// TwinCAT 3 PLC project Capannone
// ProgramVersion: 3.1.4020.10
// libraries:
//   Tc2_DALI, * (Beckhoff Automation GmbH)
//   Tc2_EnOcean, * (Beckhoff Automation GmbH)
//   Tc2_Standard, * (Beckhoff Automation GmbH)
//   Tc2_SUPS, * (Beckhoff Automation GmbH)
//   Tc2_System, * (Beckhoff Automation GmbH)
//   Tc2_TcpIp, * (Beckhoff Automation GmbH)
//   Tc2_Ulux, * (Beckhoff Automation GmbH Austria)
//   Tc2_Utilities, * (Beckhoff Automation GmbH)
//   Tc3_Module, * (Beckhoff Automation GmbH)
//   TwinCAT PLC Library ekey, * (Beckhoff Automation GmbH Austria)
//   Tc2_EIB,newest,Beckhoff Automation GmbH
//   Tc2_SerialCom,newest,Beckhoff Automation GmbH
// project tree:
//   / Clock_1Sec.TcTTO, PlcTask.TcTTO, Clock_250ms.TcTTO
//   DUTs/ Areotermo.TcDUT, struct_allarme.TcDUT, struct_allarme_1.TcDUT, Struct_Utenti.TcDUT
//   GVLs/ GVL.TcGVL, GVL_ULUX.TcGVL
//   POUs/ ADS_CX8080.TcPOU, Alarm.TcPOU, Clock_5Sec_refresh.TcPOU, Clock_2Sec_refresh_.TcPOU, DALI.TcPOU, Ekey.TcPOU, EnOcean.TcPOU, KNX.TcPOU, LUCI.TcPOU, MAIN.TcPOU, Riscaldamento.TcPOU, Timbrature.TcPOU, TIMER.TcPOU, ULUX.TcPOU
//   POUs/ProjetcFB/ Sensore_Allarme.TcPOU, Dali_arcpower_control.TcPOU, EnO_TK_SR_MDS_BAT.TcPOU, F_COIL.TcPOU, DALI_TK_SR07_rh.TcPOU, DALI_TK_SR07.TcPOU, EnO_TK_SAB05.TcPOU, EnO_TK_SR65_LI.TcPOU, Luci_Mov_Dali.TcPOU, Comando_Luce.TcPOU, Comando_LuceDali.TcPOU, Sensore_Allarme_STRU.TcPOU, Speed_Sabiana.TcPOU, ULUX_STD.TcPOU
// real-time tasks:
//   TASK 10 ms: cycle T#10ms, priority 20, ADS port 350
//   TASK Time250ms: cycle T#250ms, priority 1, ADS port 351
//   TASK Clock_1Sec: cycle T#1000ms, priority 21, ADS port 352
// I/O:
//   DEVICE Device 3 (CX-BK)
//     Box 1 (CX-BK)
//   DEVICE Device 4 (COM Port)
//   DEVICE Device 5 (RT-Ethernet Protocol), AmsNetId 192.168.60.20.6.1
//     I/O Uffici (BK9000)
//     I/O Caldaia (BK9000)
// variable links:
//   Capannone/Capannone Instance <-> Device 3 (CX-BK)/Box 1 (CX-BK)
//     Clock_1Sec Outputs/GVL.Segnale_sirena <-> Term 28 (KL2652)/Channel 2/Output
//     PlcTask Inputs/DALI.DALI_IN1/nData <-> Term 2 (KL6811)/Channel 1/Data In
//     PlcTask Inputs/DALI.DALI_IN1/nStatus <-> Term 2 (KL6811)/Channel 1/State
//     PlcTask Inputs/Ekey.ekey_in/D <-> Term 10 (KL6041)/Channel 1/Data In 0
//     PlcTask Inputs/Ekey.ekey_in/D @bit {8..168 step 8} <-> Term 10 (KL6041)/Channel 1/Data In {1..21}  (21 links)
//     PlcTask Inputs/Ekey.ekey_in/Status <-> Term 10 (KL6041)/Channel 1/State
//     PlcTask Inputs/EnOcean.enocean_in @bit 8 <-> Term 3 (KL6581)/Channel 1/Input CNODE
//     PlcTask Inputs/EnOcean.enocean_in @bit {24..48 step 8} <-> Term 3 (KL6581)/Channel 1/Input DB{0..3}  (4 links)
//     PlcTask Inputs/EnOcean.enocean_in @bit {56..80 step 8} <-> Term 3 (KL6581)/Channel 1/Input ID{0..3}  (4 links)
//     PlcTask Inputs/EnOcean.enocean_in @bit 16 <-> Term 3 (KL6581)/Channel 1/Input ORG
//     PlcTask Inputs/EnOcean.enocean_in @bit 88 <-> Term 3 (KL6581)/Channel 1/Input STATUS
//     PlcTask Inputs/EnOcean.enocean_in <-> Term 3 (KL6581)/Channel 1/Status
//     PlcTask Inputs/GVL.IN_CITOR1 <-> Term 4 (KL1809)/Channel 3/Input
//     PlcTask Inputs/GVL.IN_CITOR2 <-> Term 4 (KL1809)/Channel 2/Input
//     PlcTask Inputs/GVL.SM_C1 <-> Term 27 (KL1809)/Channel 16/Input
//     PlcTask Inputs/GVL.SM_C2 <-> Term 27 (KL1809)/Channel 15/Input
//     PlcTask Inputs/GVL.SM_C3 <-> Term 27 (KL1809)/Channel 14/Input
//     PlcTask Inputs/GVL.SM_F1 <-> Term 4 (KL1809)/Channel 6/Input
//     PlcTask Inputs/GVL.SM_F2 <-> Term 4 (KL1809)/Channel 7/Input
//     PlcTask Inputs/GVL.SM_F3 <-> Term 4 (KL1809)/Channel 8/Input
//     PlcTask Inputs/GVL.SM_F4 <-> Term 4 (KL1809)/Channel 5/Input
//     PlcTask Inputs/GVL.SM_F5 <-> Term 27 (KL1809)/Channel 2/Input
//     PlcTask Inputs/GVL.SM_R2 <-> Term 4 (KL1809)/Channel 15/Input
//     PlcTask Inputs/GVL.SM_R3 <-> Term 4 (KL1809)/Channel 16/Input
//     PlcTask Inputs/GVL.SM_R4 <-> Term 4 (KL1809)/Channel 13/Input
//     PlcTask Inputs/GVL.SM_R5 <-> Term 4 (KL1809)/Channel 14/Input
//     PlcTask Inputs/GVL.SM_S1 <-> Term 27 (KL1809)/Channel 13/Input
//     PlcTask Inputs/GVL.SM_S2 <-> Term 27 (KL1809)/Channel 8/Input
//     PlcTask Inputs/GVL.SM_U1 <-> Term 27 (KL1809)/Channel 5/Input
//     PlcTask Inputs/GVL.SM_U2 <-> Term 27 (KL1809)/Channel 6/Input
//     PlcTask Inputs/GVL.SM_U3 <-> Term 27 (KL1809)/Channel 7/Input
//     PlcTask Inputs/GVL.sens_cancello_Auto <-> Term 4 (KL1809)/Channel 9/Input
//     PlcTask Inputs/MAIN.energy_ch1_dataIN <-> Term 9 (KL3403)/Channel 1/Data In
//     PlcTask Inputs/MAIN.energy_ch2_dataIN <-> Term 9 (KL3403)/Channel 2/Data In
//     PlcTask Inputs/MAIN.energy_ch3_dataIN <-> Term 9 (KL3403)/Channel 3/Data In
//     PlcTask Inputs/MAIN.energy_ch1_state <-> Term 9 (KL3403)/Channel 1/State
//     PlcTask Inputs/MAIN.energy_ch2_state <-> Term 9 (KL3403)/Channel 2/State
//     PlcTask Inputs/MAIN.energy_ch3_state <-> Term 9 (KL3403)/Channel 3/State
//     PlcTask Inputs/MAIN.puls_chiamata <-> Term 4 (KL1809)/Channel 1/Input
//     PlcTask Outputs/DALI.DALI_OUT1/nCtrl <-> Term 2 (KL6811)/Channel 1/Ctrl
//     PlcTask Outputs/DALI.DALI_OUT1/nData <-> Term 2 (KL6811)/Channel 1/Data Out
//     PlcTask Outputs/Ekey.ekey_out/Ctrl <-> Term 10 (KL6041)/Channel 1/Ctrl
//     PlcTask Outputs/Ekey.ekey_out/D <-> Term 10 (KL6041)/Channel 1/Data Out 0
//     PlcTask Outputs/Ekey.ekey_out/D @bit {8..168 step 8} <-> Term 10 (KL6041)/Channel 1/Data Out {1..21}  (21 links)
//     PlcTask Outputs/EnOcean.enocean_out <-> Term 3 (KL6581)/Channel 1/Control
//     PlcTask Outputs/EnOcean.enocean_out @bit 8 <-> Term 3 (KL6581)/Channel 1/Output CNODE
//     PlcTask Outputs/EnOcean.enocean_out @bit {24..48 step 8} <-> Term 3 (KL6581)/Channel 1/Output DB{0..3}  (4 links)
//     PlcTask Outputs/EnOcean.enocean_out @bit {56..80 step 8} <-> Term 3 (KL6581)/Channel 1/Output ID{0..3}  (4 links)
//     PlcTask Outputs/EnOcean.enocean_out @bit 16 <-> Term 3 (KL6581)/Channel 1/Output ORG
//     PlcTask Outputs/EnOcean.enocean_out @bit 88 <-> Term 3 (KL6581)/Channel 1/Output STATUS
//     PlcTask Outputs/GVL.OUT_Pcanc_ped <-> Term 5 (KL2809)/Channel 2/Output
//     PlcTask Outputs/GVL.Sabiana{1..6}H <-> Term 12 (KL2809)/Channel {1..11 step 2}/Output  (6 links)
//     PlcTask Outputs/GVL.Sabiana{1..6}L <-> Term 12 (KL2809)/Channel {2..12 step 2}/Output  (6 links)
//     PlcTask Outputs/GVL.Segnale_radio <-> Term 28 (KL2652)/Channel 1/Output
//     PlcTask Outputs/LUCI.luci_esterne <-> Term 5 (KL2809)/Channel 5/Output
//     PlcTask Outputs/MAIN.apert_canc <-> Term 5 (KL2809)/Channel 1/Output
//     PlcTask Outputs/MAIN.compr_pistone <-> Term 5 (KL2809)/Channel 7/Output
//     PlcTask Outputs/MAIN.compr_vite <-> Term 5 (KL2809)/Channel 8/Output
//     PlcTask Outputs/MAIN.energy_ch1_control <-> Term 9 (KL3403)/Channel 1/Ctrl
//     PlcTask Outputs/MAIN.energy_ch2_control <-> Term 9 (KL3403)/Channel 2/Ctrl
//     PlcTask Outputs/MAIN.energy_ch3_control <-> Term 9 (KL3403)/Channel 3/Ctrl
//     PlcTask Outputs/MAIN.sirena_canc <-> Term 7 (KL2602)/Channel 1/Output
//   Capannone/Capannone Instance <-> Device 5 (RT-Ethernet Protocol)/I/O Caldaia (BK9000)
//     PlcTask Inputs/Riscaldamento.run_pompaprod <-> Term 39 (KL1002)/Channel 1/Input
//     PlcTask Inputs/Riscaldamento.temp_ciller <-> Term 40 (KL3204)/Channel 1/Data In
//     PlcTask Outputs/Riscaldamento.pompa_prod1 <-> Term 41 (KM2642)/Channel 1/Output
//     PlcTask Outputs/Riscaldamento.pompa_prod2 <-> Term 42 (KM2642)/Channel 2/Output
//     PlcTask Outputs/Riscaldamento.richiesta_caldaia <-> Term 42 (KM2642)/Channel 1/Output
//   Capannone/Capannone Instance <-> Device 5 (RT-Ethernet Protocol)/I/O Uffici (BK9000)
//     Clock_1Sec Outputs/GVL.Luce5 <-> Term 20 (KL2809)/Channel 5/Output
//     Clock_1Sec Outputs/GVL.Luce6 <-> Term 20 (KL2809)/Channel 6/Output
//     PlcTask Inputs/DALI.DALI_IN2/nData <-> Term 14 (KL6811)/Channel 1/Data In
//     PlcTask Inputs/DALI.DALI_IN2/nStatus <-> Term 14 (KL6811)/Channel 1/State
//     PlcTask Inputs/GVL.Th20_pompacaloreOK <-> Term 15 (KL1809)/Channel 2/Input
//     PlcTask Inputs/GVL.pulA1 <-> Term 15 (KL1809)/Channel 5/Input
//     PlcTask Inputs/GVL.pulA2 <-> Term 15 (KL1809)/Channel 3/Input
//     PlcTask Inputs/GVL.pulA3 <-> Term 15 (KL1809)/Channel 6/Input
//     PlcTask Inputs/GVL.pulA4 <-> Term 15 (KL1809)/Channel 4/Input
//     PlcTask Inputs/GVL.pulB1 <-> Term 15 (KL1809)/Channel 8/Input
//     PlcTask Inputs/GVL.pulB2 <-> Term 15 (KL1809)/Channel 7/Input
//     PlcTask Inputs/GVL.pulC1 <-> Term 15 (KL1809)/Channel 9/Input
//     PlcTask Inputs/GVL.pulD1 <-> Term 15 (KL1809)/Channel 10/Input
//     PlcTask Inputs/KNX.KNX_IN @bit {16..184 step 8} <-> Term 21 (KL6301)/Channel 1/Input Data {1..22}  (22 links)
//     PlcTask Inputs/KNX.KNX_IN <-> Term 21 (KL6301)/Channel 1/Parameter Status
//     PlcTask Outputs/DALI.DALI_OUT2/nCtrl <-> Term 14 (KL6811)/Channel 1/Ctrl
//     PlcTask Outputs/DALI.DALI_OUT2/nData <-> Term 14 (KL6811)/Channel 1/Data Out
//     PlcTask Outputs/GVL.Aer_Bagni <-> Term 20 (KL2809)/Channel 8/Output
//     PlcTask Outputs/GVL.Aer_Uffici <-> Term 20 (KL2809)/Channel 7/Output
//     PlcTask Outputs/GVL.Luce{1..4} <-> Term 20 (KL2809)/Channel {1..4}/Output  (4 links)
//     PlcTask Outputs/GVL.OUT_CILLER_ON <-> Term 19 (KL2809)/Channel 6/Output
//     PlcTask Outputs/GVL.OUT_Pingresso <-> Term 19 (KL2809)/Channel 3/Output
//     PlcTask Outputs/GVL.OUT_Pmensa <-> Term 19 (KL2809)/Channel 4/Output
//     PlcTask Outputs/GVL.out_ciller_estate <-> Term 19 (KL2809)/Channel 5/Output
//     PlcTask Outputs/KNX.KNX_OUT @bit {16..184 step 8} <-> Term 21 (KL6301)/Channel 1/Output Data {1..22}  (22 links)
//     PlcTask Outputs/KNX.KNX_OUT <-> Term 21 (KL6301)/Channel 1/Parameter Control
//     PlcTask Outputs/Riscaldamento.areotermi[10]/VHL1 <-> Term 19 (KL2809)/Channel 1/Output
//     PlcTask Outputs/Riscaldamento.areotermi[10]/VHL2 <-> Term 19 (KL2809)/Channel 2/Output
//     PlcTask Outputs/Riscaldamento.areotermi[1]/VHL1 <-> Term 16 (KL2809)/Channel 4/Output
//     PlcTask Outputs/Riscaldamento.areotermi[1]/VHL2 <-> Term 16 (KL2809)/Channel 5/Output
//     PlcTask Outputs/Riscaldamento.areotermi[2]/VHL1 <-> Term 16 (KL2809)/Channel 9/Output
//     PlcTask Outputs/Riscaldamento.areotermi[2]/VHL2 <-> Term 16 (KL2809)/Channel 10/Output
//     PlcTask Outputs/Riscaldamento.areotermi[3]/VHL1 <-> Term 16 (KL2809)/Channel 14/Output
//     PlcTask Outputs/Riscaldamento.areotermi[3]/VHL2 <-> Term 16 (KL2809)/Channel 15/Output
//     PlcTask Outputs/Riscaldamento.areotermi[4]/VHL1 <-> Term 17 (KL2809)/Channel 3/Output
//     PlcTask Outputs/Riscaldamento.areotermi[4]/VHL2 <-> Term 17 (KL2809)/Channel 4/Output
//     PlcTask Outputs/Riscaldamento.areotermi[5]/VHL1 <-> Term 17 (KL2809)/Channel 8/Output
//     PlcTask Outputs/Riscaldamento.areotermi[5]/VHL2 <-> Term 17 (KL2809)/Channel 9/Output
//     PlcTask Outputs/Riscaldamento.areotermi[6]/VHL1 <-> Term 17 (KL2809)/Channel 13/Output
//     PlcTask Outputs/Riscaldamento.areotermi[6]/VHL2 <-> Term 17 (KL2809)/Channel 14/Output
//     PlcTask Outputs/Riscaldamento.areotermi[7]/VHL1 <-> Term 18 (KL2809)/Channel 2/Output
//     PlcTask Outputs/Riscaldamento.areotermi[7]/VHL2 <-> Term 18 (KL2809)/Channel 3/Output
//     PlcTask Outputs/Riscaldamento.areotermi[8]/VHL1 <-> Term 18 (KL2809)/Channel 7/Output
//     PlcTask Outputs/Riscaldamento.areotermi[8]/VHL2 <-> Term 18 (KL2809)/Channel 8/Output
//     PlcTask Outputs/Riscaldamento.areotermi[9]/VHL1 <-> Term 18 (KL2809)/Channel 12/Output
//     PlcTask Outputs/Riscaldamento.areotermi[9]/VHL2 <-> Term 18 (KL2809)/Channel 13/Output
//     PlcTask Outputs/Riscaldamento.areotermi[10]/speed1 <-> Term 18 (KL2809)/Channel 14/Output
//     PlcTask Outputs/Riscaldamento.areotermi[10]/speed2 <-> Term 18 (KL2809)/Channel 15/Output
//     PlcTask Outputs/Riscaldamento.areotermi[10]/speed3 <-> Term 18 (KL2809)/Channel 16/Output
//     PlcTask Outputs/Riscaldamento.areotermi[1]/speed1 <-> Term 16 (KL2809)/Channel 1/Output
//     PlcTask Outputs/Riscaldamento.areotermi[1]/speed2 <-> Term 16 (KL2809)/Channel 2/Output
//     PlcTask Outputs/Riscaldamento.areotermi[1]/speed3 <-> Term 16 (KL2809)/Channel 3/Output
//     PlcTask Outputs/Riscaldamento.areotermi[2]/speed1 <-> Term 16 (KL2809)/Channel 6/Output
//     PlcTask Outputs/Riscaldamento.areotermi[2]/speed2 <-> Term 16 (KL2809)/Channel 7/Output
//     PlcTask Outputs/Riscaldamento.areotermi[2]/speed3 <-> Term 16 (KL2809)/Channel 8/Output
//     PlcTask Outputs/Riscaldamento.areotermi[3]/speed1 <-> Term 16 (KL2809)/Channel 11/Output
//     PlcTask Outputs/Riscaldamento.areotermi[3]/speed2 <-> Term 16 (KL2809)/Channel 12/Output
//     PlcTask Outputs/Riscaldamento.areotermi[3]/speed3 <-> Term 16 (KL2809)/Channel 13/Output
//     PlcTask Outputs/Riscaldamento.areotermi[4]/speed1 <-> Term 16 (KL2809)/Channel 16/Output
//     PlcTask Outputs/Riscaldamento.areotermi[4]/speed2 <-> Term 17 (KL2809)/Channel 1/Output
//     PlcTask Outputs/Riscaldamento.areotermi[4]/speed3 <-> Term 17 (KL2809)/Channel 2/Output
//     PlcTask Outputs/Riscaldamento.areotermi[5]/speed1 <-> Term 17 (KL2809)/Channel 5/Output
//     PlcTask Outputs/Riscaldamento.areotermi[5]/speed2 <-> Term 17 (KL2809)/Channel 6/Output
//     PlcTask Outputs/Riscaldamento.areotermi[5]/speed3 <-> Term 17 (KL2809)/Channel 7/Output
//     PlcTask Outputs/Riscaldamento.areotermi[6]/speed1 <-> Term 17 (KL2809)/Channel 10/Output
//     PlcTask Outputs/Riscaldamento.areotermi[6]/speed2 <-> Term 17 (KL2809)/Channel 11/Output
//     PlcTask Outputs/Riscaldamento.areotermi[6]/speed3 <-> Term 17 (KL2809)/Channel 12/Output
//     PlcTask Outputs/Riscaldamento.areotermi[7]/speed1 <-> Term 17 (KL2809)/Channel 15/Output
//     PlcTask Outputs/Riscaldamento.areotermi[7]/speed2 <-> Term 17 (KL2809)/Channel 16/Output
//     PlcTask Outputs/Riscaldamento.areotermi[7]/speed3 <-> Term 18 (KL2809)/Channel 1/Output
//     PlcTask Outputs/Riscaldamento.areotermi[8]/speed1 <-> Term 18 (KL2809)/Channel 4/Output
//     PlcTask Outputs/Riscaldamento.areotermi[8]/speed2 <-> Term 18 (KL2809)/Channel 5/Output
//     PlcTask Outputs/Riscaldamento.areotermi[8]/speed3 <-> Term 18 (KL2809)/Channel 6/Output
//     PlcTask Outputs/Riscaldamento.areotermi[9]/speed1 <-> Term 18 (KL2809)/Channel 9/Output
//     PlcTask Outputs/Riscaldamento.areotermi[9]/speed2 <-> Term 18 (KL2809)/Channel 10/Output
//     PlcTask Outputs/Riscaldamento.areotermi[9]/speed3 <-> Term 18 (KL2809)/Channel 11/Output

CONFIGURATION Capannone
    RESOURCE PLC ON TwinCAT3
        TASK Clock_1Sec(INTERVAL := T#1000ms, PRIORITY := 21);
        TASK PlcTask(INTERVAL := T#10ms, PRIORITY := 20);
        TASK Clock_250ms(INTERVAL := T#250ms, PRIORITY := 1);
        PROGRAM Clock_5Sec_refresh WITH Clock_1Sec : Clock_5Sec_refresh;
        PROGRAM Clock_2Sec_refresh_ WITH Clock_1Sec : Clock_2Sec_refresh_;
        PROGRAM MAIN WITH PlcTask : MAIN;
        PROGRAM Timbrature WITH PlcTask : Timbrature;
        PROGRAM TIMER WITH Clock_250ms : TIMER;
    END_RESOURCE
END_CONFIGURATION

// ---- DUTs/Areotermo.TcDUT
TYPE Areotermo :
STRUCT
	speed1:BOOL;
	speed2:BOOL;
	speed3:BOOL;
	VHL1:BOOL;
	VHL2:BOOL;
END_STRUCT
END_TYPE

// ---- DUTs/struct_allarme.TcDUT
TYPE struct_allarme :
STRUCT
	mode_a0 : BOOL:=TRUE;
	mode_a1 : BOOL;
	mode_a2 : BOOL;
	mode_a3 : BOOL;
	mode_a4 : BOOL;
	delay_allarme : TIME:= T#30S;
	allarme_dis : BOOL;
	sens_mov : BOOL;
	porta_fin : BOOL;
	sensore : BOOL;
	sens_ritardato : BOOL;
	sens_attivo : BOOL;
END_STRUCT
END_TYPE

// ---- DUTs/struct_allarme_1.TcDUT
TYPE struct_allarme_1 :
STRUCT
	sens_zonaA: BOOL;
	sens_zonaB: BOOL;
	sens_zonaC: BOOL;
	sens_zonaD: BOOL;
	ritardo_ON: TIME; //Ritardo accensione sensore in secondi
	ritardo_OFF: TIME; //Ritardo spegnimento sensore in secondi
	HMI_Ritardo_ON: REAL; //HMI ritardo accensione sensore
	HMI_Ritardo_OFF: REAL; //HMI ritardo spegnimento sensore
	sens_ON_OFF: BOOL; //Accensione/spegnimento sensore TRUE=acceso FALSE= spento
	allarme_sensore: BOOL; //Segnale uscita allarme sensore
	tamper_sensore: BOOL; //Segnale uscita tamper sensore
	stato_sensore: BYTE; //0=OFF 1=allarme generato 2=tamper 3=in allarme attivo ma libero 4=in allarme attivo 5=acceso libero 6=acceso occupato
	testo_sensore: STRING; //Nome e funzione sensore
	sensore_preallarme: BOOL; //Segnale sonoro con allarme attivo
END_STRUCT
END_TYPE

// ---- DUTs/Struct_Utenti.TcDUT
TYPE Struct_Utenti :
STRUCT
	user_type: BYTE;
	num_badge: STRING;
	nome_utente: STRING;
END_STRUCT
END_TYPE

// ---- GVLs/GVL.TcGVL
VAR_GLOBAL
	//cancella
	AAA_Prova1: BOOL;
	//EnOcean
	enocean_buffer: STR_KL6581;
	//DALI
	DALI_BUFFER1: ST_DALIV2CommandBuffer; //Comando luci capannone
	DALI_BUFFER2: ST_DALIV2CommandBuffer; //Comando luci uffici
	//Ekey
	ekey_scanner_cancello: FB_EKEY_FingerScanner; //Numero di serie ekey cancello:31160073
	ekey_scanner_produzione: FB_EKEY_FingerScanner; //Numero di serie ekey produzione:24180820 vecchio:37160686
	ekey_scanner_ingresso: FB_EKEY_FingerScanner;//Numero di serie ekey ingresso:37160693 vecchio:37160693
	HMI_finger: BOOL;
	HMI_finger_RFID: BOOL;
	HMI_userRFID: BYTE;
	apri_file: FB_FileOpen;
	inserisci_testo: fb_fileputs;
	chiudi_file: fb_fileclose;
	indice_utente: INT:=1;
	Nmu: BYTE:=30; //Numero massimo utenti
	hmi_utentesu: BOOL; //Pulsante indice utente i più
	hmi_utentegiu: BOOL; //Pulsante indice utente i meno
	HMI_save_utente: BOOL; //Salva parametri utenti su HMI
	HMI_annulla: BOOL; // Annulla cambio dati utente
	HMI_user_type: BYTE;
	HMI_num_badge: STRING;
	HMI_nome_utente: STRING;
	//ULUX
	ulux_buffer: ST_ULUX_COMMANDBUFFER;
	//KNX
	RAIN: BOOL;
	Temp_OUTSIDE: REAL;
	wind_speed: REAL;
	LUX_OUTSIDEF: REAL;
	LUX_OUTSIDER: REAL;
	LUX_OUTSIDEL: REAL;
	knx_p1: BOOL;
	knx_p2: BOOL;
	knx_p3: BOOL;
	knx_p4: BOOL;
	Temp_INSIDE: REAL;
	stato_temp: BOOL; //Stato sensore temperatura 0=OK 1=Difettoso
	
	//ALLARME
	alarm_Service: BOOL;
	allarme_on: BOOL;
	sensori_mov: ARRAY [1..30] OF sensore_allarme;
	mode_A: BYTE; //Modalità inserimento allarme valori da 0 a 4
	test_Sirena: BOOL;
	test_radio: BOOL;
	allarme_memreset: BOOL;
	stringa_allarme: STRING;
	stringa_2_allarme: STRING; //Stringa di visualizzazione in file di testo allarmi
	sensori_STRU: ARRAY [0..30] OF sensore_allarme_STRU;
	ingresso_sens AT %I*: ARRAY [0..30] OF BOOL; //Array segnale fisico sensore
	reset_tamper: BOOL;
	reset_allarme: BOOL;
	manutenzione_sensore: BOOL;
	
	//CILLER
	out_ciller_estate AT %Q*: BOOL;
	OUT_CILLER_ON AT %Q*: BOOL;
	//PORTE
	OUT_Pingresso AT %Q*: BOOL;
	OUT_Pmensa AT %Q*: BOOL;
	OUT_Pcanc_ped AT %Q*: BOOL;
	IN_CITOR1 AT %I*: BOOL;
	IN_CITOR2 AT %I*: BOOL;
	//ALTRO
	tempo: BOOL;
	count: INT;
	ora_plc: nt_gettime;
	tempo_ulux: timestruct;
	aggiorna: BYTE; //Variabile timer
	orario: STRING;
	orario_2: STRING;
	giorni_sett: BOOL;
	Read_Puls1: FB_Rec_RPS_Switch;
	HMI_ctrl_allarme: BOOL;
	sens_cancello_Auto AT %I*: BOOL;
	hmi_cancello: BOOL;
	HMI_compressore_2: BOOL;
	HMI_currentL1: WORD;
	HMI_currentL2: WORD;
	HMI_currentL3: WORD;
	HMI_voltageL1: WORD;
	HMI_voltageL2: WORD;
	HMI_voltageL3: WORD;
	HMI_powerL1: WORD;
	HMI_powerL2: WORD;
	HMI_powerL3: WORD;
	HMI_energyL1: WORD;
	HMI_energyL2: WORD;
	HMI_energyL3: WORD;
	HMI_frequencyL1: WORD;
	HMI_frequencyL2: WORD;
	HMI_frequencyL3: WORD;
	HMI_Allarme: BOOL;
	HMI_luci_on: ARRAY [0..6] OF BOOL; //Luci uffici ON
	HMI_luci_off: ARRAY [0..6] OF BOOL; //Luci uffici OFF
	HMI_cond: ARRAY [0..6] OF INT;
	HMI_luce1: BOOL; //Comando luce bagno 1 da HMI
	HMI_luce2: BOOL; //Comando luce bagno 2 da HMI
	HMI_luce_3: BOOL; //Comando luci esterne da HMI
	HMI_luce4: BOOL; //Comando luce ripostiglio da HMI
	HMI_luce_server: BOOL; //Comando luce server da HMI
	HMI_luce_lstamp: BOOL; //Comando luce locale stampante
	HMI_luce_offRD: BOOL; //Comando luce officina R&D
	
	light_soft: BOOL;
	Light_on: BOOL;
	Light_off: BOOL;
	dali_power_off: BOOL;
	Sabiana1L AT %Q*: BOOL; //Sabiana 1 Low Speed
	Sabiana1H AT %Q*: BOOL; //Sabiana 1 High Speed
	Sabiana2L AT %Q*: BOOL; //Sabiana 2 Low Speed
	Sabiana2H AT %Q*: BOOL; //Sabiana 2 High Speed
	Sabiana3L AT %Q*: BOOL; //Sabiana 3 Low Speed
	Sabiana3H AT %Q*: BOOL; //Sabiana 3 High Speed
	Sabiana4L AT %Q*: BOOL; //Sabiana 4 Low Speed
	Sabiana4H AT %Q*: BOOL; //Sabiana 4 High Speed
	Sabiana5L AT %Q*: BOOL; //Sabiana 5 Low Speed
	Sabiana5H AT %Q*: BOOL; //Sabiana 5 High Speed
	Sabiana6L AT %Q*: BOOL; //Sabiana 6 Low Speed
	Sabiana6H AT %Q*: BOOL; //Sabiana 6 High Speed
	
	HMI_SabianaManCTRL : ARRAY [1..6] OF BYTE; //Controllo Manuale Sabiana
	HMI_PompaProd : BOOL; //Comando Manuale da pannello pompa riscaldamento produzione
	TempZ0:UINT; //Temperatura zona 0 - Capannone
	TempZ1:UINT; //Temperatura zona 1 - Ingresso
	TempZ2:UINT; //Temperatura zona 2 - Amministrazione
	TempZ3:UINT; //Temperatura zona 3 - Direzione
	TempZ4:UINT; //Temperatura zona 4 - Sala Riunioni
	TempZ5:UINT; //Temperatura zona 5 - Uffico Tecnico
	TempZ6:UINT; //Temperatura zona 6 - Ufficio Produzione
	TempZ7:UINT; //Temperatura zona 7 - Locale Svago
	ConONz1:INT; //Condizionatore ON/OFF zona 1
	ConONz2:INT; //Condizionatore ON/OFF zona 2
	ConONz3:INT; //Condizionatore ON/OFF zona 3
	ConONz4:INT; //Condizionatore ON/OFF zona 4
	ConONz5:INT; //Condizionatore ON/OFF zona 5
	ConONz6:INT; //Condizionatore ON/OFF zona 6
	ConONz7:INT; //Condizionatore ON/OFF zona 7
	HMI_Umidita:BYTE; //Umidità Capannone
	Th20_CaldaiaOK (*AT %I**):BOOL:=TRUE; //Temperatura H20 Caldaia OK x aria
	Th20_pompacaloreOK AT %I*:BOOL; //Temperatura H20 Pompa Calore OK x aria
	SensoreSez1 : BOOL; (*Sensore Apertura Sezionale 1*)
	SensoreSez2 : BOOL; (*Sensore Apertura Sezionale 2*)
	Luce1 AT %Q*:BOOL; (*Relè Luci BAGNO UFFICI 1*)
	Luce2 AT %Q*:BOOL; (*Relè Luci BAGNO UFFICI 2*)
	Luce3 AT %Q*:BOOL; (*Relè Luci esterno ENTRATA*)
	Luce4 AT %Q*:BOOL; (*Relè Luci RIPOSTIGLIO*)
	Luce5 AT %Q*:BOOL; (*Relè Luci 1*)
	Luce6 AT %Q*:BOOL; (*Relè Luci 1*)
	Aer_Uffici AT %Q*:BOOL; (*Relè Luci 1*)
	Aer_Bagni AT %Q* :BOOL; (*Areazione Bagno*)
	time_now: UINT;
	GuestIN_OK: BOOL;
	UserIN_OK: BOOL;
	HMI_blink: BOOL; //Bit per blink su HMI
	luci_ufficio_off: BOOL;
	//Pulsantiera A
	pulA1 AT %I* :BOOL;
	pulA2 AT %I* :BOOL;
	pulA3 AT %I* :BOOL;
	pulA4 AT %I* :BOOL;
	//Pulsantiera B
	pulB1 AT %I* :BOOL;
	pulB2 AT %I* :BOOL;
	//Pulsantiera C
	pulC1 AT %I* :BOOL;
	//Pulsantiera D
	pulD1 AT %I* :BOOL;
	prod_summer_fan: INT;
	meetingroom_active: BOOL;
	//Sensori di movimento
	SM_F1 AT %I*: BOOL;
	SM_F2 AT %I*: BOOL;
	SM_F3 AT %I*: BOOL;
	SM_F4 AT %I*: BOOL;
	SM_F5 AT %I*: BOOL;
	SM_S1 AT %I*: BOOL;
	SM_S2 AT %I*: BOOL;
	(*SM_R1 AT %I*: BOOL;
	SM_R2 AT %I*: BOOL;
	SM_R3 AT %I*: BOOL;
	SM_R4 AT %I*: BOOL;
	SM_R5 AT %I*: BOOL;
	SM_D1 AT %I*: BOOL;*)
	SM_C1 AT %I*: BOOL;
	//SM_C2 AT %I*: BOOL;
	//SM_C3 AT %I*: BOOL;
	SM_U1 AT %I*: BOOL; //Sensore Ufficio Tecnico
	SM_U2 AT %I*: BOOL; //Sensore Locale Svago
	//SM_U3 AT %I*: BOOL; //Sensore Ingresso
	Tamper_interno AT %I*: BOOL;
	Tamper_fronte AT %I*: BOOL;
	Tamper_retro AT %I*: BOOL;
	Tamper_sinistro AT %I*: BOOL;
	Segnale_radio AT %Q*: BOOL;
	Segnale_sirena AT %Q*: BOOL;
	
	OFFICE_vhac_MODE:BYTE; //0= ESTATE - 1 INVERNO PDC - 2 INVERNO MISTO
	gruppo8_arc_level: BYTE;
	gruppo9_arc_level: BYTE;
	//Telecamere
	camera_index: INT;
	HMI_blink_2: BOOL;
	HMI_Cancelletto: BOOL;
	HMI_porta: BOOL;
	camera_counter: INT;
	str_camera1: STRING(255);
	camera1: STRING(255);
	camera2: STRING(255);
	camera3: STRING(255);
	camera4: STRING(255);
	//Comando luci bagno produzione e spogliatoi
	count_bagno_prod: INT;
	timer_bagno_prod: TP;
	pulse_bagno_prod: TP;
	luce_bagni: FB_Send_RPS_SwitchAuto;
	luce_spogliatoio: FB_Send_RPS_SwitchAuto;
	MOVIMENTO_BAGNO_PROD: EnO_TK_SR_MDS_BAT;
	RITARDO_LUCE_BAGNO_PROD: TOF;
	
	variable_update: BOOL := FALSE;
	aggiorna_sec: BOOL;
END_VAR
VAR_GLOBAL RETAIN PERSISTENT
	ON:BOOL := TRUE;
	var_ora_trasp: BOOL;
	var_ora_dip: BOOL;
	user_type: ARRAY [1..30] OF BYTE;
	utenti: ARRAY [1..30] OF struct_utenti;
	allarme: BOOL;
	allarme_Attivo: BYTE; //0=OFF 1=Gruppo A 2=Gruppo B 3=Gruppo C 4=Gruppo D
	HMI_sirena: BOOL; //Per ON-OFF segnale sirena da HMI
	HMI_radio: BOOL; //Per ON-OFF segnale radio da HMI
	delay_allarme_on: TIME:=T#150S;
	delay_sirena_off: TIME:=T#2M;
	time_IN1:UINT:=0630;
	time_OUT1:UINT:=1300;
	time_IN2:UINT:=1300;
	time_out2:UINT:=1800;
	time_work_IN1:UINT:=0800;
	time_work_OUT1:UINT:=1230;
	time_work_IN2:UINT:=1330;
	time_work_OUT2:UINT:=1700;
	saturday_work:BOOL;
	holidays:BOOL;
	auto_allarm: BOOL:=TRUE;
	HeatingdMode : BYTE := 2; (*Modo funzionamento riscaldamento 0= OFF - 1=MAN - 2=AUTO - 3=Estate*)
	OFFICE_VHAC_EI:BOOL; (*0=INVERNO 1=ESTATE*)
	estate: BOOL;
	inverno: BOOL;
	HMI_TEMPprod : UINT:=170; (*Temperatura di riferimento PRODUZIONE*)
	HMI_TEMPuff : ARRAY [1..7] OF UINT; //Array temperatura di riferimento UFFICI tec. e prod. è la stessa
	HMI_var_tempuff : ARRAY [1..7] OF UINT; //Array variazione temperatura ambiente UFFICI
	HMI_TEMPuff_max: UINT:=280; //Temperatura di riferimento massima UFFICI
	HMI_TEMPuff_min: UINT:=240; //Temperatura di riferimento minima UFFICI
	HMI_luci_capannone: BYTE:=250; (*Luminosità luci capannone*)
	luci_capannone_aut: BOOL:=TRUE;
	sens_allarme: ARRAY [1..30] OF struct_allarme;
	sens_allarme_stru: ARRAY [0..30] OF struct_allarme_1; //Array struttura sensori
	tamper AT %I*: ARRAY [0..30] OF BOOL; //Array segnale tamper sensore
	alarm_history: ARRAY [1..50] OF STRING;
	warning_history: ARRAY [1..50] OF STRING;
	
	TempOffSabiana1: INT:=450; (*Temperatura Ciller OFF x Sabiana*)
	TempOffSabiana2: INT:=450; (*Temperatura Ciller OFF x Sabiana*)
	TempOffSabiana3: INT:=650; (*Temperatura Ciller OFF x Sabiana*)
	TempOffSabiana4: INT:=550; (*Temperatura Ciller OFF x Sabiana*)
	TempOffSabiana5: INT:=450; (*Temperatura Ciller OFF x Sabiana*)
	TempOffSabiana6: INT:=600; (*Temperatura Ciller OFF x Sabiana*)
END_VAR

// ---- GVLs/GVL_ULUX.TcGVL
(* Automatic generated on 16/02/2017 16.07.46 from u::Lux Config V1.34.635, Build 2474 *)
(* u::Lux Projectfile: C:\Users\ACO\Documents\OWNCLOUD\Software PLC\00 - DOMOTICA\4 - ULUX\Programma_Uffici.uLux *)

(* VarNameEndings: *)
(* _IP: IP-Address of a Control or a Switch *)
(* _ID: ID of an Actor or a Switch *)
(* _EDITVALUE: EditValue of an Actor *)
(* _OUTPUT: Output of an Actor *)
(* _INPUT: Input of an Actor *)

VAR_GLOBAL CONSTANT
	(* Common Constants *)
	PROJEKT_ULUX_CONTROL_IP:STRING:='192.168.60.120';
	PROJEKT_ULUX_CONTROL_AMSNETID:STRING:= '5.29.125.252.1.1';

	(* Constants for u::Lux Switch Design_Ingresso *)
	ULUX_SWITCH_DESIGN_INGRESSO_ULUX_SWITCH_INGRESSO_ID:WORD:=1;

	(* Constants for u::Lux Switch Design_Ingresso\Attori_Ingresso *)
	ATTORI_INGRESSO_ONOFF_LUCE_ID:WORD:=1;
	ATTORI_INGRESSO_DIMMER_ID:WORD:=2;
	ATTORI_INGRESSO_HEIZUNG_TEMPERATUR_ID:WORD:=3;
	ATTORI_INGRESSO_ACTOR_4_ID:WORD:=4;
	ATTORI_INGRESSO_COND_ONOFF_ID:WORD:=5;
	ATTORI_INGRESSO_ACTOR_6_ID:WORD:=6;
	ATTORI_INGRESSO_ACTOR_7_ID:WORD:=7;
	ATTORI_INGRESSO_ACTOR_8_ID:WORD:=8;
	ATTORI_INGRESSO_ACTOR_9_ID:WORD:=9;
	ATTORI_INGRESSO_ACTOR_10_ID:WORD:=10;

	(* Constants for u::Lux Switch Design_Amministrazione *)
	ULUX_SWITCH_DESIGN_AMMINISTRAZIONE_ULUX_SWITCH_AMMINISTRAZIONE_ID:WORD:=2;

	(* Constants for u::Lux Switch Design_Amministrazione\Attori_Amministrazione *)
	ATTORI_AMMINISTRAZIONE_ONOFF_LUCE_ID:WORD:=11;
	ATTORI_AMMINISTRAZIONE_DIMMER_ID:WORD:=12;
	ATTORI_AMMINISTRAZIONE_HEIZUNG_TEMPERATUR_ID:WORD:=13;
	ATTORI_AMMINISTRAZIONE_ACTOR_4_ID:WORD:=14;
	ATTORI_AMMINISTRAZIONE_COND_ONOFF_ID:WORD:=15;
	ATTORI_AMMINISTRAZIONE_ACTOR_6_ID:WORD:=16;
	ATTORI_AMMINISTRAZIONE_ACTOR_7_ID:WORD:=17;
	ATTORI_AMMINISTRAZIONE_ACTOR_8_ID:WORD:=18;
	ATTORI_AMMINISTRAZIONE_ACTOR_9_ID:WORD:=19;
	ATTORI_AMMINISTRAZIONE_ACTOR_10_ID:WORD:=20;

	(* Constants for u::Lux Switch Design_Direzione *)
	ULUX_SWITCH_DESIGN_DIREZIONE_ULUX_SWITCH_DIREZIONE_ID:WORD:=3;

	(* Constants for u::Lux Switch Design_Direzione\Attori_Direzione *)
	ATTORI_DIREZIONE_ONOFF_LUCE_ID:WORD:=21;
	ATTORI_DIREZIONE_DIMMER_ID:WORD:=22;
	ATTORI_DIREZIONE_HEIZUNG_TEMPERATUR_ID:WORD:=23;
	ATTORI_DIREZIONE_ACTOR_4_ID:WORD:=24;
	ATTORI_DIREZIONE_COND_ONOFF_ID:WORD:=25;
	ATTORI_DIREZIONE_ACTOR_6_ID:WORD:=26;
	ATTORI_DIREZIONE_ACTOR_7_ID:WORD:=27;
	ATTORI_DIREZIONE_ACTOR_8_ID:WORD:=28;
	ATTORI_DIREZIONE_ACTOR_9_ID:WORD:=29;
	ATTORI_DIREZIONE_ACTOR_10_ID:WORD:=30;

	(* Constants for u::Lux Switch Design_Sala_Riunioni *)
	ULUX_SWITCH_DESIGN_SALA_RIUNIONI_ULUX_SWITCH_SALA_RIUNIONI_ID:WORD:=4;

	(* Constants for u::Lux Switch Design_Sala_Riunioni\Attori_Sala_Riunioni *)
	ATTORI_SALA_RIUNIONI_ONOFF_LUCE_ID:WORD:=31;
	ATTORI_SALA_RIUNIONI_DIMMER_ID:WORD:=32;
	ATTORI_SALA_RIUNIONI_HEIZUNG_TEMPERATUR_ID:WORD:=33;
	ATTORI_SALA_RIUNIONI_ACTOR_4_ID:WORD:=34;
	ATTORI_SALA_RIUNIONI_COND_ONOFF_ID:WORD:=35;
	ATTORI_SALA_RIUNIONI_ACTOR_6_ID:WORD:=36;
	ATTORI_SALA_RIUNIONI_ACTOR_7_ID:WORD:=37;
	ATTORI_SALA_RIUNIONI_ACTOR_8_ID:WORD:=38;
	ATTORI_SALA_RIUNIONI_ACTOR_9_ID:WORD:=39;
	ATTORI_SALA_RIUNIONI_ACTOR_10_ID:WORD:=40;

	(* Constants for u::Lux Switch Design_Tecnico *)
	ULUX_SWITCH_DESIGN_TECNICO_ULUX_SWITCH_TECNICO_ID:WORD:=5;

	(* Constants for u::Lux Switch Design_Tecnico\Attori_Tecnico *)
	ATTORI_TECNICO_ONOFF_LUCE_ID:WORD:=41;
	ATTORI_TECNICO_DIMMER_ID:WORD:=42;
	ATTORI_TECNICO_HEIZUNG_TEMPERATUR_ID:WORD:=43;
	ATTORI_TECNICO_ACTOR_4_ID:WORD:=44;
	ATTORI_TECNICO_COND_ONOFF_ID:WORD:=45;
	ATTORI_TECNICO_ACTOR_6_ID:WORD:=46;
	ATTORI_TECNICO_ACTOR_7_ID:WORD:=47;
	ATTORI_TECNICO_ACTOR_8_ID:WORD:=48;
	ATTORI_TECNICO_ACTOR_9_ID:WORD:=49;
	ATTORI_TECNICO_ACTOR_10_ID:WORD:=50;

	(* Constants for u::Lux Switch Design_Produzione *)
	ULUX_SWITCH_DESIGN_PRODUZIONE_ULUX_SWITCH_PRODUZIONE_1_ID:WORD:=6;

	(* Constants for u::Lux Switch Design_Produzione\Attori_Produzione *)
	ATTORI_PRODUZIONE_ONOFF_LUCE_ID:WORD:=51;
	ATTORI_PRODUZIONE_DIMMER_ID:WORD:=52;
	ATTORI_PRODUZIONE_HEIZUNG_TEMPERATUR_ID:WORD:=53;
	ATTORI_PRODUZIONE_ACTOR_4_ID:WORD:=54;
	ATTORI_PRODUZIONE_COND_ONOFF_ID:WORD:=55;
	ATTORI_PRODUZIONE_ACTOR_6_ID:WORD:=56;
	ATTORI_PRODUZIONE_ACTOR_7_ID:WORD:=57;
	ATTORI_PRODUZIONE_ACTOR_8_ID:WORD:=58;
	ATTORI_PRODUZIONE_ACTOR_9_ID:WORD:=59;
	ATTORI_PRODUZIONE_ACTOR_10_ID:WORD:=60;

	(* Constants for u::Lux Switch Design_Locale_Svago *)
	ULUX_SWITCH_DESIGN_LOCALE_SVAGO_ULUX_SWITCH_LOCALE_SVAGO_ID:WORD:=7;

	(* Constants for u::Lux Switch Design_Locale_Svago\Attori_Locale Svago *)
	ATTORI_LOCALE_SVAGO_ONOFF_LUCE_ID:WORD:=61;
	ATTORI_LOCALE_SVAGO_DIMMER_ID:WORD:=62;
	ATTORI_LOCALE_SVAGO_HEIZUNG_TEMPERATUR_ID:WORD:=63;
	ATTORI_LOCALE_SVAGO_ACTOR_4_ID:WORD:=64;
	ATTORI_LOCALE_SVAGO_COND_ONOFF_ID:WORD:=65;
	ATTORI_LOCALE_SVAGO_ACTOR_6_ID:WORD:=66;
	ATTORI_LOCALE_SVAGO_ACTOR_7_ID:WORD:=67;
	ATTORI_LOCALE_SVAGO_ACTOR_8_ID:WORD:=68;
	ATTORI_LOCALE_SVAGO_ACTOR_9_ID:WORD:=69;
	ATTORI_LOCALE_SVAGO_ACTOR_10_ID:WORD:=70;

	(* Number of Switches and Controls *)
	ULUXSWITCH_COUNT:WORD:=7;
	ULUXPLC_COUNT:WORD:=1;
END_VAR

VAR_GLOBAL
	(* Structure for u::Lux Switches *)
	ULUX_CMD_BUFFER: ST_ULUX_COMMANDBUFFER;

	(* Common Values *)

	(* Values for u::Lux Switch Design_Ingresso *)
	ULUX_SWITCH_DESIGN_INGRESSO_ULUX_SWITCH_INGRESSO_IP:STRING;

	(* Values for u::Lux Switch Design_Ingresso\Attori_Ingresso *)

	(* Values for u::Lux Switch Design_Amministrazione *)
	ULUX_SWITCH_DESIGN_AMMINISTRAZIONE_ULUX_SWITCH_AMMINISTRAZIONE_IP:STRING;

	(* Values for u::Lux Switch Design_Amministrazione\Attori_Amministrazione *)

	(* Values for u::Lux Switch Design_Direzione *)
	ULUX_SWITCH_DESIGN_DIREZIONE_ULUX_SWITCH_DIREZIONE_IP:STRING;

	(* Values for u::Lux Switch Design_Direzione\Attori_Direzione *)

	(* Values for u::Lux Switch Design_Sala_Riunioni *)
	ULUX_SWITCH_DESIGN_SALA_RIUNIONI_ULUX_SWITCH_SALA_RIUNIONI_IP:STRING;

	(* Values for u::Lux Switch Design_Sala_Riunioni\Attori_Sala_Riunioni *)

	(* Values for u::Lux Switch Design_Tecnico *)
	ULUX_SWITCH_DESIGN_TECNICO_ULUX_SWITCH_TECNICO_IP:STRING;

	(* Values for u::Lux Switch Design_Tecnico\Attori_Tecnico *)

	(* Values for u::Lux Switch Design_Produzione *)
	ULUX_SWITCH_DESIGN_PRODUZIONE_ULUX_SWITCH_PRODUZIONE_1_IP:STRING;
	ULUX_SWITCH_DESIGN_PRODUZIONE_ULUX_SWITCH_PRODUZIONE_2_IP:STRING;

	(* Values for u::Lux Switch Design_Produzione\Attori_Produzione *)

	(* Values for u::Lux Switch Design_Locale_Svago *)
	ULUX_SWITCH_DESIGN_LOCALE_SVAGO_ULUX_SWITCH_LOCALE_SVAGO_IP:STRING;

	(* Values for u::Lux Switch Design_Locale_Svago\Attori_Locale Svago *)

END_VAR

VAR_GLOBAL PERSISTENT
	(* Common Values *)

	(* Values for u::Lux Switch Design_Ingresso *)

	(* Values for u::Lux Switch Design_Ingresso\Attori_Ingresso *)
	ATTORI_INGRESSO_ONOFF_LUCE_EDITVALUE:BOOL;
	ATTORI_INGRESSO_ONOFF_LUCE_OUTPUT AT %Q*:BOOL;
	ATTORI_INGRESSO_DIMMER_EDITVALUE:BOOL;
	ATTORI_INGRESSO_DIMMER_OUTPUT AT %Q*:BOOL;

	(* Values for u::Lux Switch Design_Amministrazione *)

	(* Values for u::Lux Switch Design_Amministrazione\Attori_Amministrazione *)
	ATTORI_AMMINISTRAZIONE_ONOFF_LUCE_EDITVALUE:BOOL;
	ATTORI_AMMINISTRAZIONE_ONOFF_LUCE_OUTPUT AT %Q*:BOOL;
	ATTORI_AMMINISTRAZIONE_DIMMER_EDITVALUE:BOOL;
	ATTORI_AMMINISTRAZIONE_DIMMER_OUTPUT AT %Q*:BOOL;

	(* Values for u::Lux Switch Design_Direzione *)

	(* Values for u::Lux Switch Design_Direzione\Attori_Direzione *)
	ATTORI_DIREZIONE_ONOFF_LUCE_EDITVALUE:BOOL;
	ATTORI_DIREZIONE_ONOFF_LUCE_OUTPUT AT %Q*:BOOL;
	ATTORI_DIREZIONE_DIMMER_EDITVALUE:BOOL;
	ATTORI_DIREZIONE_DIMMER_OUTPUT AT %Q*:BOOL;

	(* Values for u::Lux Switch Design_Sala_Riunioni *)

	(* Values for u::Lux Switch Design_Sala_Riunioni\Attori_Sala_Riunioni *)
	ATTORI_SALA_RIUNIONI_ONOFF_LUCE_EDITVALUE:BOOL;
	ATTORI_SALA_RIUNIONI_ONOFF_LUCE_OUTPUT AT %Q*:BOOL;
	ATTORI_SALA_RIUNIONI_DIMMER_EDITVALUE:BOOL;
	ATTORI_SALA_RIUNIONI_DIMMER_OUTPUT AT %Q*:BOOL;

	(* Values for u::Lux Switch Design_Tecnico *)

	(* Values for u::Lux Switch Design_Tecnico\Attori_Tecnico *)
	ATTORI_TECNICO_ONOFF_LUCE_EDITVALUE:BOOL;
	ATTORI_TECNICO_ONOFF_LUCE_OUTPUT AT %Q*:BOOL;
	ATTORI_TECNICO_DIMMER_EDITVALUE:BOOL;
	ATTORI_TECNICO_DIMMER_OUTPUT AT %Q*:BOOL;

	(* Values for u::Lux Switch Design_Produzione *)

	(* Values for u::Lux Switch Design_Produzione\Attori_Produzione *)
	ATTORI_PRODUZIONE_ONOFF_LUCE_EDITVALUE:BOOL;
	ATTORI_PRODUZIONE_ONOFF_LUCE_OUTPUT AT %Q*:BOOL;
	ATTORI_PRODUZIONE_DIMMER_EDITVALUE:BOOL;
	ATTORI_PRODUZIONE_DIMMER_OUTPUT AT %Q*:BOOL;

	(* Values for u::Lux Switch Design_Locale_Svago *)

	(* Values for u::Lux Switch Design_Locale_Svago\Attori_Locale Svago *)
	ATTORI_LOCALE_SVAGO_ONOFF_LUCE_EDITVALUE:BOOL;
	ATTORI_LOCALE_SVAGO_ONOFF_LUCE_OUTPUT AT %Q*:BOOL;
	ATTORI_LOCALE_SVAGO_DIMMER_EDITVALUE:BOOL;
	ATTORI_LOCALE_SVAGO_DIMMER_OUTPUT AT %Q*:BOOL;

END_VAR

// ---- POUs/Clock_5Sec_refresh.TcPOU
PROGRAM Clock_5Sec_refresh
VAR
	timer:INT;
END_VAR

timer:=timer+1;
IF timer=10 THEN
	timer:=0;
END_IF
IF timer <5 THEN
	HMI_blink:=FALSE;
ELSE 
	HMI_blink:=TRUE;
END_IF

END_PROGRAM

// ---- POUs/TIMER.TcPOU
PROGRAM TIMER
VAR
	i: INT;
	Delay_on: TON;
	stps: TIME:=T#1S;
	aggiorna1s: INT; //Aggiorna timer 1s
	timer_1s: BOOL;
END_VAR

// aggiorna variabili generali
aggiorna:=aggiorna+1;
IF aggiorna=(i*2) THEN
	aggiorna:=0;
END_IF
IF aggiorna<i THEN
	aggiorna_sec:=TRUE;
ELSE
	aggiorna_sec:=FALSE;
END_IF
//Timer 1s
aggiorna1s:=aggiorna1s+1;
IF aggiorna1s>=4 THEN
	aggiorna1s:=0;
	timer_1s:=TRUE;
ELSE
	timer_1s:=FALSE;
END_IF
ora_plc(
	NETID:= , 
	START:=timer_1s, 
	TMOUT:= T#2S, 
	BUSY=> , 
	ERR=> , 
	ERRID=> , 
	TIMESTR=> );

//Tempo dispositivi ulux
tempo_ulux.wHour:=ORA_PLC.TIMESTR.wHour;
tempo_ulux.wMinute:=ORA_PLC.TIMESTR.wMinute;
tempo_ulux.wSecond:=ORA_PLC.TIMESTR.wSecond;
tempo_ulux.wDay:=ORA_PLC.TIMESTR.wDay;
tempo_ulux.wMonth:=ORA_PLC.TIMESTR.wMonth;
tempo_ulux.wYear:=ORA_PLC.TIMESTR.wYear;

//Impulso 1 clock con settaggio variabile
Delay_on(IN:= TRUE AND NOT delay_on.Q, PT:= stps, Q=> , ET=> );

IF delay_on.Q THEN
	camera_counter:=camera_counter+1;
END_IF;
camera1:=concat('http://192.168.60.109/snap.jpeg?cb=',INT_TO_STRING(camera_counter));
camera2:=concat('http://192.168.60.105/snap.jpeg?cb=',INT_TO_STRING(camera_counter));
camera3:=concat('http://192.168.60.113/snap.jpeg?cb=',INT_TO_STRING(camera_counter));
camera4:=concat('http://192.168.60.111/snap.jpeg?cb=',INT_TO_STRING(camera_counter));

END_PROGRAM

// ---- POUs/Clock_2Sec_refresh_.TcPOU
PROGRAM Clock_2Sec_refresh_
VAR
	timer:INT;
END_VAR

timer:=timer+1;
IF timer=4 THEN
	timer:=0;
END_IF
IF timer < 2 THEN
	HMI_blink_2:=TRUE;
ELSE 
	HMI_blink_2:=FALSE;
END_IF

END_PROGRAM

// ---- POUs/MAIN.TcPOU
PROGRAM MAIN
VAR
	SAVE_RETAIN: FB_S_UPS_CX51x0;
	puls_chiamata AT %I*: BOOL;
	sirena_canc AT %Q*: BOOL;
	apert_canc AT %Q*: BOOL;
	Sirena_cancello: TP;
	apertura_porta_ingr: TP;
	apert_canc1 : BOOL; //Apertura cancello per trasportatori
	apert_canc2 : BOOL; //Apertura cancello per dipendenti
	apert_canc3 : BOOL; //Apertura cancello con sensore e con allarme
	compr_pistone AT %Q* : BOOL;
	compr_vite AT %Q* : BOOL;
	luce : ARRAY [1..10] OF comando_luce;
	
	//controllo Energia
	energy_ch1_control AT %Q* : USINT;
	energy_ch2_control AT %Q* : USINT;
	energy_ch3_control AT %Q* : USINT;
	energy_ch1_dataIN AT %I* : INT;
	energy_ch2_dataIN AT %I* : INT;
	energy_ch3_dataIN AT %I* : INT;
	energy_ch1_state AT %I* : USINT;
	energy_ch2_state AT %I* : USINT;
	energy_ch3_state AT %I* : USINT;
	energy_function:INT;
	
	//Tempo_Cancello_trasp: RS;
	//Tempo_Cancello_Dip: RS;
	Entrata_Trasp: TP;
	timer_allarme: TON;
	Energydata_update: R_TRIG;
	alarm_counter: INT;
	Accensione_luci: F_TRIG;
	Spegnimento_luci: R_TRIG;
	Delay_allarme: TON;
	led_allarmeon: BOOL;
	ins_allarme: R_TRIG;
	ins_AUTOallarme: F_TRIG;
	allarme_off: R_TRIG;
	puls_allarme: TON;
	HMI_puls_allarme: TON; //Inserimento allarme da pannello
END_VAR

//ads_CX8080();
enocean();
DALI();
Ekey();
RISCALDAMENTO();
luci();
ULUX();
KNX();
Alarm();
// Salvataggio dati con UPS Interno
SAVE_RETAIN(
	sNetID:= '', 
	iPLCPort:= 851, 
	iUPSPort:= , 
	tTimeout:= , 
	eUpsMode:= , 
	ePersistentMode:= , 
	tRecoverTime:= , 
	bPowerFailDetect=> , 
	eState=> );

(*Gestione e Conversione ORA*)
time_now := (ORA_PLC.TIMESTR.wHour*100)+ ora_plc.TIMESTR.wMinute;
(*Gestione Orari GUEST*)
GuestIN_OK:= ((time_now>=time_work_IN1 AND time_now<=time_work_OUT1)
			OR (time_now>=time_work_IN2 AND time_now<=time_work_OUT2))
			AND allarme_Attivo=0;
(*Gestione Orari USER*)
IF holidays OR ora_plc.TIMESTR.wDayOfWeek=0 THEN
	USERIN_OK:=FALSE;
ELSIF (ora_plc.TIMESTR.wDayOfWeek=6 AND saturday_work) AND (time_now>=time_IN1 AND time_now<=time_OUT1) THEN
	USERIN_OK:=TRUE;
ELSIF (ora_plc.TIMESTR.wDayOfWeek>=1 AND ora_plc.TIMESTR.wDayOfWeek<=5) AND ((time_now>=time_IN1 AND time_now<=time_OUT1)
																		OR (time_now>=time_IN2 AND time_now<=time_OUT2)) THEN
	USERIN_OK:=TRUE;
ELSE
	USERIN_OK:=FALSE;	
END_IF
(*Segnale allarme*)
(*allarme_off(CLK:= time_now=0730, Q=> );
IF allarme_off.Q THEN
	allarme:=FALSE;
END_IF*)
//Inserimento allarme con pulsante a muro o HMI
puls_allarme(IN:= puld1, PT:= T#5S, Q=> , ET=> );
HMI_puls_allarme(IN:= HMI_Allarme, PT:= T#5S, Q=> , ET=> );
IF puls_allarme.Q OR hmi_puls_allarme.Q THEN
	allarme_Attivo:=1;
END_IF
ins_allarme(CLK:= time_now=1730, Q=> );
ins_AUTOallarme(CLK:= time_now=1730, Q=> );
IF ins_allarme.Q AND auto_allarm THEN
	allarme_Attivo:=1;
END_IF
IF ins_AUTOallarme.Q THEN
	auto_allarm:=TRUE;
END_IF
luce[1].pulsante:=TRUE;
//Compressori
compr_vite:=TRUE;
compr_pistone:=allarme_Attivo=0;

//--> GESTIONE CANCELLO
//Apertura cancello per tipo utente per dipendenti + spegnimento allarme
IF ekey_scanner_cancello.bGoodFinger AND utenti[ekey_scanner_cancello.byRecUserID].user_type=3 THEN
	apert_canc2:=TRUE;
	allarme_attivo:=0;
ELSIF ekey_scanner_cancello.bGoodFinger AND utenti[ekey_scanner_cancello.byRecUserID].user_type=0 AND userin_OK THEN
	apert_canc2:=TRUE;
	allarme_Attivo:=0;
ELSE
	apert_canc2:=FALSE;
END_IF
//Spegnimento allarme con scanner ingresso
IF ekey_scanner_ingresso.bGoodFinger AND utenti[ekey_scanner_cancello.byRecUserID].user_type=3 THEN
	allarme_Attivo:=0;
END_IF
//Spegnimento allarme automatico con scanner ingresso per pulizia
IF ekey_scanner_ingresso.bGoodFinger AND ekey_scanner_ingresso.byRecUserID=26 AND allarme_Attivo=0 AND time_now<1730 THEN
	auto_allarm:=FALSE;
END_IF
//Apertura porta ingresso con ekey e HMI
apertura_porta_ingr(IN:= (ekey_scanner_ingresso.bGoodFinger AND allarme_Attivo=0) OR HMI_porta, PT:= T#1S, Q=> out_Pingresso, ET=> );
//Apertura cancello con pulsante per trasportatori
IF puls_chiamata AND guestin_ok THEN
	apert_canc1:=TRUE;
ELSE
	apert_canc1:=FALSE;
END_IF
//Apertura cancello con sensore auto e con allarme
timer_allarme(IN:= allarme_Attivo<>0, PT:= delay_allarme_on, Q=> , ET=> );
apert_canc3:=NOT timer_Allarme.Q AND sens_cancello_auto;

apert_canc:=apert_canc1 OR apert_canc2 OR apert_canc3 OR hmi_cancello OR IN_CITOR1;
Sirena_cancello(IN:= puls_chiamata, PT:= T#5S, Q=> sirena_canc, ET=> );

//Apertura cancello pedonale
OUT_Pcanc_ped:=IN_CITOR2 OR HMI_Cancelletto;
//<-- GESTIONE CANCELLO

//Controllo Energia	
CASE energy_function OF
	0:	energy_ch1_control :=0;
		IF energy_ch1_control=energy_ch1_state THEN
			HMI_currentL1:=energy_ch1_dataIN;
			energy_function:=energy_function+1;
		END_IF;
	1:	energy_ch2_control :=0;
		IF energy_ch2_control=energy_ch2_state THEN
			HMI_currentL2:=energy_ch2_dataIN;
			energy_function:=energy_function+1;
		END_IF;
	2:	energy_ch3_control :=0;
		IF energy_ch3_control=energy_ch3_state THEN
			HMI_currentL3:=energy_ch3_dataIN;
			energy_function:=energy_function+1;
		END_IF;
	3:	energy_ch1_control :=1;
		IF energy_ch1_control=energy_ch1_state THEN
			HMI_voltageL1:=energy_ch1_dataIN;
			energy_function:=energy_function+1;
		END_IF;
	4:	energy_ch2_control :=1;
		IF energy_ch2_control=energy_ch2_state THEN
			HMI_voltageL2:=energy_ch2_dataIN;
			energy_function:=energy_function+1;
		END_IF;
	5:	energy_ch3_control :=1;
		IF energy_ch3_control=energy_ch3_state THEN
			HMI_voltageL3:=energy_ch3_dataIN;
			energy_function:=energy_function+1;
		END_IF;	
	6:	energy_ch1_control :=2;
		IF energy_ch1_control=energy_ch1_state THEN
			HMI_PowerL1:=energy_ch1_dataIN;
			energy_function:=energy_function+1;
		END_IF;
	7:	energy_ch2_control :=2;
		IF energy_ch2_control=energy_ch2_state THEN
			HMI_PowerL2:=energy_ch2_dataIN;
			energy_function:=energy_function+1;
		END_IF;
	8:	energy_ch3_control :=2;
		IF energy_ch3_control=energy_ch3_state THEN
			HMI_PowerL3:=energy_ch3_dataIN;
			energy_function:=energy_function+1;
		END_IF;	
	9:	energy_ch1_control :=4;
		IF energy_ch1_control=energy_ch1_state THEN
			HMI_energyL1:=energy_ch1_dataIN;
			energy_function:=energy_function+1;
		END_IF;
	10:	energy_ch2_control :=4;
		IF energy_ch2_control=energy_ch2_state THEN
			HMI_energyL2:=energy_ch2_dataIN;
			energy_function:=energy_function+1;
		END_IF;
	11:	energy_ch3_control :=4;
		IF energy_ch3_control=energy_ch3_state THEN
			HMI_energyL3:=energy_ch3_dataIN;
			energy_function:=energy_function+1;
		END_IF;	
	12:	energy_ch1_control :=8;
		IF energy_ch1_control=energy_ch1_state THEN
			HMI_frequencyL1:=energy_ch1_dataIN;
			energy_function:=energy_function+1;
		END_IF;
	13:	energy_ch2_control :=8;
		IF energy_ch2_control=energy_ch2_state THEN
			HMI_frequencyL2:=energy_ch2_dataIN;
			energy_function:=energy_function+1;
		END_IF;
	14:	energy_ch3_control :=8;
		IF energy_ch3_control=energy_ch3_state THEN
			HMI_frequencyL3:=energy_ch3_dataIN;
			energy_function:=0;
		END_IF;	
END_CASE;

ACTION ACT:
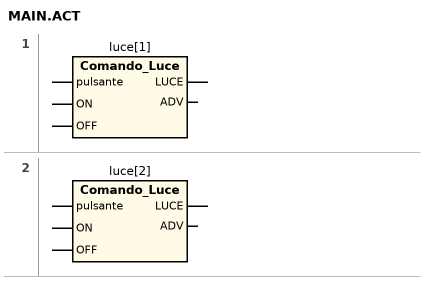
// NETWORK 1
luce[1](); // Comando_Luce

// NETWORK 2
luce[2](); // Comando_Luce
END_ACTION

END_PROGRAM

// ---- POUs/ProjetcFB/Comando_Luce.TcPOU
FUNCTION_BLOCK Comando_Luce
VAR_INPUT
	pulsante: BOOL;
	ON:BOOL;
	OFF:BOOL;
END_VAR
VAR_OUTPUT
	LUCE: BOOL;
	ADV:BOOL;
END_VAR
VAR
	livello_luce: BYTE;
	pulsa: R_TRIG;
	advanced_function: TON;
	adv_Rtrig: R_TRIG;
END_VAR

pulsa(CLK:= pulsante, Q=> );
IF pulsa.Q AND luce THEN
	luce:=FALSE;
ELSIF pulsa.Q AND NOT luce THEN
	luce:=TRUE;
END_IF;
IF on THEN
	luce:=TRUE;
END_IF
IF OFF THEN
	luce:=FALSE;
END_IF
advanced_function(IN:=pulsante , PT:=T#2S, Q=> , ET=> );
adv_Rtrig(CLK:=advanced_function.Q , Q=>adv );

END_FUNCTION_BLOCK

// ---- POUs/EnOcean.TcPOU
PROGRAM EnOcean
VAR
	Enocean_comm: FB_KL6581;
	enocean_in AT %I*: KL6581_Input;
	enocean_out AT %Q*: KL6581_Output;
	Enocean_Search: FB_EnOcean_Search;
	Sens_mov_spogliatoio: FB_Rec_Generic;
	
	movimento_Spogliatoio: BOOL;
	trigger_mov_spogliatoio: R_TRIG;
	trigger_mov_bagni: R_TRIG;
	timer_luce_spogliatoio: TOF;
	on_luce_spogliatoio: R_TRIG;
	off_luce_spogliatoio: F_TRIG;
	
	test2: BOOL;
	test1: BOOL;
	Spogliatoio: EnO_TK_SAB05;
	Bagno_prod1: EnO_TK_SAB05;
	puls_bagno_prod: FB_Rec_RPS_Switch;

	puls_porta_fumatori: FB_Rec_RPS_Switch;
	search: BOOL;
	
	MOVIMENTO_RIPOSTIGLIO: EnO_TK_SR_MDS_BAT;
	MOVIMENTO_BAGNOU1: EnO_TK_SR_MDS_BAT;
	puls_bagno_U2: FB_Rec_RPS_Switch;
	MOVIMENTO_BAGNOU2: EnO_TK_SR_MDS_BAT;
	
	RITARDO_LUCE_RIPOSTIGLIO: TOF;
	RITARDO_LUCE_BAGNOU1: TOF;
	RITARDO_LUCE_BAGNOU2: TOF;
	
	puls_ventilazione: FB_Rec_RPS_Switch;
	puls_ingr_1: FB_Rec_RPS_Switch;
	puls_ingr_2: FB_Rec_RPS_Switch;
	puls_ingr_3: FB_Rec_RPS_Switch;
	luce_enocean_1: Dali_arcpower_control;
	comando_luce_1: Comando_LuceDali;
	gruppo_enocean_0: Dali_arcpower_control;
	comando_gruppo_0: Comando_LuceDali;
	VentilazioneProduzioneSU: R_TRIG;
	VentilazioneProduzioneGIU: R_TRIG;
	VentilazioneProduzionegii: BOOL;
	
	puls_locale_stamp: FB_Rec_RPS_Switch;
	luce_lstamp_ON: R_TRIG;
	luce_lstamp_OFF: R_TRIG;
	puls_officina_RD: FB_Rec_RPS_Switch;
	luce_offRD_ON: R_TRIG;
	luce_offRD_OFF: R_TRIG;

	timer_luce_bagno: TON;
	timer_luce_bagno2: TON;
END_VAR

//Comunicazione EnOcean
Enocean_comm(
	bInit:= TRUE, 
	nIdx:= 1, 
	bReady=> , 
	bBusy=> , 
	bError=> , 
	iErrorID=> , 
	str_KL6581=> enocean_buffer, 
	stKL6581_in:= enocean_in, 
	stKL6581_out:= enocean_out);
//Ricerca dispositivo EnOcean
Enocean_Search(
	bStart:= search, 
	str_KL6581:= enocean_buffer, 
	byNode:= , 
	bReceive=> , 
	iDevices=> , 
	ar_ID=> );
//Lettura pulsante 1
Read_Puls1(
	str_KL6581:= enocean_buffer, 
	byNode:= , 
	dw_ID:= 1415876,
	str_EnOceanSwitch=> , 
	by_Node=> , 
	bReceive=> );
(*//Sensore movimento
Sens_mov_spogliatoio(
	str_KL6581:= enocean_buffer, 
	byNode:= 1, 
	
	dw_ID:= 16#01920C34(*16#0191F8D2*),
	ar_Value=> , 
	by_Node=> , 
	by_STATE=> , 
	bReceive=> , 
	EnOceanTyp=> );
movimento_spogliatoio:=sens_mov_Spogliatoio.ar_Value[1]>127;
(*movimento_spogliatoio:=sens_mov_Spogliatoio.ar_Value[0]=13;*)
on_luce_spogliatoio(CLK:=movimento_spogliatoio AND NOT timer_luce_spogliatoio.Q , Q=> );
timer_luce_spogliatoio(IN:=movimento_Spogliatoio , PT:= T#1S, Q=> , ET=> );
off_luce_spogliatoio(CLK:=timer_luce_spogliatoio.Q , Q=> );*)

//Pulsante luci bagno produzione
puls_bagno_prod(
	str_KL6581:= enocean_buffer, 
	byNode:= , 
	dw_ID:= 16#002A4D65, 
	str_EnOceanSwitch=> , 
	by_Node=> , 
	bReceive=> );
	
//Comando luci bagno produzione e spogliatoi
//timer_bagno_prod(IN:= puls_bagno_prod.str_EnOceanSwitch.bT2_ON OR puls_bagno_prod.str_EnOceanSwitch.bT2_OFF, PT:= T#310S, Q=> , ET=> );
//pulse_bagno_prod(IN:= MOVIMENTO_BAGNO_PROD.Moviment, PT:= T#310S, Q=> , ET=> );
MOVIMENTO_BAGNO_PROD(ID:=16#01A357A7 , BAT_KO=> , LUX=> , Moviment=> );
RITARDO_LUCE_BAGNO_PROD(IN:=MOVIMENTO_BAGNO_PROD.Moviment , PT:=T#1m , Q=> , ET=> );

luce_spogliatoio(
	bStart:= puls_bagno_prod.str_EnOceanSwitch.bT2_ON, 
	bData:= , 
	by_Node:= 1, 
	t_SwitchDelay:= T#0S, 
	nRockerID:= 0, 
	nEnOceanID:=12 , 
	str_KL6581:= enocean_buffer, 
	bBusy=> , 
	bError=> , 
	iErrorID=> );
luce_bagni(
	bStart:= puls_bagno_prod.str_EnOceanSwitch.bT2_OFF,
	bData:= , 
	by_Node:= 1, 
	t_SwitchDelay:= T#0S, 
	nRockerID:= 0, 
	nEnOceanID:= 11, 
	str_KL6581:= enocean_buffer, 
	bBusy=> , 
	bError=> , 
	iErrorID=> );

//Pulsante apertura porta fumatori
puls_porta_fumatori(
	str_KL6581:= enocean_buffer, 
	byNode:= , 
	dw_ID:= 16#008B627F, 
	str_EnOceanSwitch=> , 
	by_Node=> , 
	bReceive=> );
IF puls_porta_fumatori.str_EnOceanSwitch.bT1_OFF OR puls_porta_fumatori.str_EnOceanSwitch.bT1_ON OR puls_porta_fumatori.str_EnOceanSwitch.bT2_OFF OR puls_porta_fumatori.str_EnOceanSwitch.bT2_ON AND allarme_Attivo=0 THEN
	out_pmensa:=TRUE;
ELSE
	out_pmensa:=FALSE;
END_IF

(*Bagni Servizio*)
Spogliatoio(
	IDr:= (*16#0188D643*) , 
	IDw:= 20, 
	bsend:= , 
	t_setpoint:= , 
	b_SB:= , 
	b_RIN:= , 
	b_LFS:= , 
	b_VO:= , 
	b_VC:= );

(*Bagno_prod1(
	IDr:=16#0188D441, 
	IDw:= 21, 
	bsend:= , 
	t_setpoint:= , 
	b_SB:= , 
	b_RIN:= , 
	b_LFS:= , 
	b_VO:= , 
	b_VC:= );*)

(*//Ventilatori produzione
puls_ventilazione(
	str_KL6581:= enocean_buffer, 
	byNode:= , 
	dw_ID:= 16#002A4D49, 
	str_EnOceanSwitch=> , 
	by_Node=> , 
	bReceive=> );
VentilazioneProduzioneSU(CLK:=puls_ventilazione.str_EnOceanSwitch.bT2_ON , Q=> );
VentilazioneProduzioneGIU(CLK:=puls_ventilazione.str_EnOceanSwitch.bT2_OFF , Q=> );
	IF VentilazioneProduzioneSU.Q THEN
		prod_summer_fan:=prod_summer_fan+1;
			IF prod_summer_fan=3 THEN
				prod_summer_fan:=0;
			END_IF
	END_IF
	IF VentilazioneProduzionegiu.Q THEN
		prod_summer_fan:=prod_summer_fan-1;
			IF prod_summer_fan=-1 THEN
				prod_summer_fan:=2;
			END_IF
	END_IF*)
IF allarme_Attivo<>0 THEN
	prod_summer_fan:=0;
END_IF

//Pulsante luci locale stampante
puls_locale_stamp(
	str_KL6581:= enocean_buffer, 
	byNode:= , 
	dw_ID:= 16#002A4D53, 
	str_EnOceanSwitch=> , 
	by_Node=> , 
	bReceive=> );
luce_lstamp_ON(CLK:=puls_locale_stamp.str_EnOceanSwitch.bT2_ON , Q=> );
luce_lstamp_OFF(CLK:=puls_locale_stamp.str_EnOceanSwitch.bT2_OFF , Q=> );
IF  luce_lstamp_ON.Q THEN
	hmi_luce_lstamp:=TRUE;
END_IF
IF luce_lstamp_OFF.Q THEN
	hmi_luce_lstamp:=FALSE;
END_IF
IF hmi_luce_lstamp THEN
	gruppo8_arc_level:=254;
ELSE
	gruppo8_arc_level:=0;
END_IF
IF allarme_Attivo<>0 THEN
	gruppo8_arc_level:=0;
	hmi_luce_lstamp:=FALSE;
END_IF

//Pulsante luci officina R&D
puls_officina_RD(
	str_KL6581:= enocean_buffer, 
	byNode:= , 
	dw_ID:= 16#002A4D48, 
	str_EnOceanSwitch=> , 
	by_Node=> , 
	bReceive=> );
luce_offRD_ON(CLK:=puls_officina_RD.str_EnOceanSwitch.bT2_ON , Q=> );
luce_offRD_OFF(CLK:=puls_officina_RD.str_EnOceanSwitch.bT2_OFF , Q=> );
IF luce_offrd_on.Q THEN
	hmi_luce_offrd:=TRUE;
END_IF
IF luce_offrd_off.Q THEN
	hmi_luce_offrd:=FALSE;
END_IF
IF hmi_luce_offRD THEN
	gruppo9_arc_level:=254;
ELSE
	gruppo9_arc_level:=0;
END_IF
IF allarme_attivo<>0 THEN
	gruppo9_arc_level:=0;
	hmi_luce_offRD:=FALSE;
END_IF
	
//RIPOSTIGLIO
MOVIMENTO_RIPOSTIGLIO(ID:=16#01A35725 , BAT_KO=> , LUX=> , Moviment=> );
RITARDO_LUCE_RIPOSTIGLIO(IN:= MOVIMENTO_RIPOSTIGLIO.Moviment OR HMI_luce4, PT:= T#3M, Q=> LUCE4, ET=> );
//BAGNO 1 UFFICI
MOVIMENTO_BAGNOU1(ID:=16#00061F66 , BAT_KO=> , LUX=> , Moviment=> );
RITARDO_LUCE_BAGNOU1(IN:= puls_bagno_U2.str_EnOceanSwitch.bT2_ON OR MOVIMENTO_BAGNOU1.Moviment OR HMI_luce1, PT:= T#5M, Q=> luce1, ET=> );
//BAGNO 2 UFFICI
puls_bagno_U2(
	str_KL6581:= enocean_buffer, 
	byNode:= , 
	dw_ID:= 16#002A4D49, 
	str_EnOceanSwitch=> , 
	by_Node=> , 
	bReceive=> );
MOVIMENTO_BAGNOU2(ID:=16#01A32DA5 , BAT_KO=> , LUX=> , Moviment=> );
RITARDO_LUCE_BAGNOU2(IN:= puls_bagno_U2.str_EnOceanSwitch.bT2_ON OR MOVIMENTO_BAGNOU2.Moviment OR HMI_LUCE2, PT:= T#5M, Q=> LUCE2, ET=> );
//AREAZIONE BAGNI
AER_BAGNI:=LUCE1 OR LUCE2;
//PULSANTE 1 INGRESSO
puls_ingr_1(
	str_KL6581:= enocean_buffer, 
	byNode:= , 
	dw_ID:= 16#0088F11C, 
	str_EnOceanSwitch=> , 
	by_Node=> , 
	bReceive=> );
luce_enocean_1(light_level:= , ADDR:= 1, MODE:= 0, daliBuffer:= dali_buffer2);
comando_luce_1(
	pulsante:= , 
	ON:= puls_ingr_1.str_EnOceanSwitch.bT1_off, 
	OFF:= puls_ingr_1.str_EnOceanSwitch.bT1_On, 
	up:= puls_ingr_1.str_EnOceanSwitch.bT2_Off, 
	down:= puls_ingr_1.str_EnOceanSwitch.bT2_On, 
	light_level=> luce_enocean_1.light_level, 
	ADV=> );
//PULSANTE 2 INGRESSO
puls_ingr_2(
	str_KL6581:= enocean_buffer, 
	byNode:= , 
	dw_ID:= 16#002A4C9A, 
	str_EnOceanSwitch=> , 
	by_Node=> , 
	bReceive=> );
//PULSANTE 3 INGRESSO
puls_ingr_3(
	str_KL6581:= enocean_buffer, 
	byNode:= , 
	dw_ID:= 16#008C2463, 
	str_EnOceanSwitch=> , 
	by_Node=> , 
	bReceive=> );
gruppo_enocean_0(light_level:= , ADDR:= 0, MODE:= 1, daliBuffer:= dali_buffer2);
comando_gruppo_0(
	pulsante:= , 
	ON:= puls_ingr_3.str_EnOceanSwitch.bT1_OFF, 
	OFF:= puls_ingr_3.str_EnOceanSwitch.bT1_on, 
	up:= puls_ingr_3.str_EnOceanSwitch.bT2_OFF, 
	down:= puls_ingr_3.str_EnOceanSwitch.bT2_ON, 
	light_level=> gruppo_enocean_0.light_level, 
	ADV=> );

END_PROGRAM

// ---- POUs/ProjetcFB/EnO_TK_SAB05.TcPOU
FUNCTION_BLOCK EnO_TK_SAB05
VAR_INPUT
	IDr : DWORD;
	IDw : BYTE;
	bsend:BOOL;
	t_setpoint:BYTE;
	b_SB:BOOL; //Summer bit, reduction of energy cnsumption
	b_RIN:BOOL; //Run init Sequence
	b_LFS:BOOL; // Lift SET Inizialization, adjustment to the valve stroke
	b_VO:BOOL; // Valve Open - Maintenance
	b_VC:BOOL; // Valve Closed
END_VAR
VAR_OUTPUT
	CV:BYTE;//Curent Value;
	TMP:BYTE;//Temperature;
	LRNB:BOOL;// LRN Bit
END_VAR
VAR
	READ: FB_Rec_Generic;
	WRITE: FB_Send_Generic;
	byte1:WORD;
	data: DWORD;
	byte3:DWORD;
END_VAR

READ(
	str_KL6581:=enocean_buffer , 
	byNode:=1 , 
	dw_ID:=IDr , 
	ar_Value=> , 
	by_Node=> , 
	by_STATE=> , 
	bReceive=> , 
	EnOceanTyp=> );
	
cv:=read.ar_Value[3];
TMP:=read.ar_Value[1];
LRNB:=read.ar_Value[0].3;

byte3:=DINT_TO_BYTE (TRUNC(t_setpoint*6.375));
byte1.2:=TRUE; //set point selection (0..40°C)
byte1.3:=b_SB; 
byte1.4:=b_VC; 
byte1.5:=b_VO; 
byte1.6:=b_LFS; 
byte1.7:=b_RIN; 

data:=(SHL(byte3,16))+(SHL(byte1,8));

WRITE(
	bStart:= bsend, 
	by_Node:=1 , 
	by_ORG:= , 
	pt_SendData:= ADR(data) , 
	by_STATE:= , 
	nEnOceanID:=IDw , 
	str_KL6581:= enocean_buffer , 
	bBusy=> , 
	bError=> , 
	iErrorID=> );

END_FUNCTION_BLOCK

// ---- POUs/ProjetcFB/EnO_TK_SR_MDS_BAT.TcPOU
FUNCTION_BLOCK EnO_TK_SR_MDS_BAT
VAR_INPUT
	ID:DWORD;
END_VAR
VAR_OUTPUT
	BAT_KO:BOOL;
	LUX:WORD;
	Moviment:BOOL;
END_VAR
VAR
	Read: FB_Rec_Generic;
END_VAR

Read(
	str_KL6581:= enocean_buffer, 
	byNode:=1 , 
	dw_ID:= ID, 
	ar_Value=> , 
	by_Node=> , 
	by_STATE=> , 
	bReceive=> , 
	EnOceanTyp=> );
	
MOviment:=NOT read.ar_Value[0].1;
IF read.ar_Value[3]<120 THEN
	bat_KO:=TRUE;
ELSE
	bat_KO:=FALSE;
END_IF
LUX:=read.ar_Value[2]*2;

END_FUNCTION_BLOCK

// ---- POUs/ProjetcFB/Dali_arcpower_control.TcPOU
FUNCTION_BLOCK Dali_arcpower_control
VAR_INPUT
	light_level:BYTE; // VALUE FROM 85 TO 254 ADMITTED
	ADDR:BYTE; //INDIRIZZO DALI DA COMANDARE
	MODE: E_DALIV2AddrType; //TIPO DI COMANDO DA MANDARE 0=SINGOLO NODO - 1= GROUP - 2 - BROADCAST
END_VAR
VAR_OUTPUT
END_VAR
VAR_IN_OUT
	daliBuffer:ST_DALIV2CommandBuffer;
END_VAR
VAR
	arcpower: FB_DALIV2DirectArcPowerControl;
	light_level_temp:BYTE;
END_VAR

IF light_level<>light_level_temp THEN
	arcpower.bStart:=TRUE;
	light_level_temp:=light_level;
ELSE 
	arcpower.bStart:=FALSE;
END_IF
arcpower(
	bStart:= , 
	nAddr:= ADDR, 
	eAddrType:=MODE , 
	eCommandPriority:= , 
	nArcPowerLevel:=light_level , 
	bBusy=> , 
	bError=> , 
	nErrorId=> , 
	stCommandBuffer:=daliBuffer);

END_FUNCTION_BLOCK

// ---- POUs/ProjetcFB/Comando_LuceDali.TcPOU
FUNCTION_BLOCK Comando_LuceDali
VAR_INPUT
	pulsante AT %I*: BOOL;
	ON AT %I*:BOOL;
	OFF AT %I*:BOOL;
	up AT %I*:BOOL;
	down at %I*:BOOL;
END_VAR
VAR_OUTPUT
	light_level: BYTE;
	ADV:BOOL;
END_VAR
VAR
	livello_luce: BYTE;
	pulsa: R_TRIG;
	advanced_function: TON;
	adv_Rtrig: R_TRIG;
	luce:BOOL;
	level: word;
END_VAR

pulsa(CLK:= pulsante, Q=> );
IF pulsa.Q AND luce THEN
	luce:=FALSE;
ELSIF pulsa.Q AND NOT luce THEN
	luce:=TRUE;
END_IF;
IF on THEN
	luce:=TRUE;
END_IF
IF OFF THEN
	luce:=FALSE;
END_IF
advanced_function(IN:=pulsante , PT:=T#2S, Q=> , ET=> );
adv_Rtrig(CLK:=advanced_function.Q , Q=>adv );

IF level<2540 AND up AND luce THEN
	level:=level+1;
ELSIF level>840 AND down AND luce THEN
	level:=level-1;
END_IF

IF luce OR ON THEN
	light_level:=REAL_TO_BYTE(TRUNC(level/10));
ELSIF NOT luce OR OFF THEN
	 light_level:=0;
END_IF

END_FUNCTION_BLOCK

// ---- POUs/DALI.TcPOU
PROGRAM DALI
VAR
	DALI_COMM1: FB_DALIV2Communication;	
	DALI_IN1 AT %I*: ST_DALIV2InData;
	DALI_OUT1 AT %Q*: ST_DALIV2OutData;
	DALI_COMM2: FB_DALIV2Communication;
	DALI_IN2 AT %I*: ST_DALIV2InData;
	DALI_OUT2 AT %Q*: ST_DALIV2OutData;
	DALI_POWER_1: FB_DALIV2DirectArcPowerControl;
	LAMP_1_OFF: FB_DALIV2Off;
	office_POWER_1: FB_DALIV2DirectArcPowerControl;
	office_OFF: FB_DALIV2Off;
	all_on: BOOL;
	naddr_on: byte;
	start_lighton: BOOL;
	arcpowerlevel: BYTE := 80;
	light_ON_delay: BYTE;
	dali_power_start: BOOL;
	
	Level_LuceServer: Luci_Mov_Dali;
	Comando_diretto: FB_DALIV2DirectArcPowerControl;
END_VAR

DALI_COMM1(
	bResetMaximumDemandCounter:= , 
	bResetOverflowCounter:= , 
	arrBufferDemandMeter=> , 
	arrBufferMaximumDemandMeter=> , 
	arrBufferOverflowCounter=> , 
	bLineIsBusy=> , 
	bLineIsInitialized=> , 
	stDALIInData:=DALI_IN1, 
	stDALIOutData:= DALI_OUT1, 
	stCommandBuffer:= DALI_BUFFER1);
	
DALI_COMM2(
	bResetMaximumDemandCounter:= , 
	bResetOverflowCounter:= , 
	arrBufferDemandMeter=> , 
	arrBufferMaximumDemandMeter=> , 
	arrBufferOverflowCounter=> , 
	bLineIsBusy=> , 
	bLineIsInitialized=> , 
	stDALIInData:=DALI_IN2, 
	stDALIOutData:= DALI_OUT2, 
	stCommandBuffer:= DALI_BUFFER2);

//comando manuale luce
comando_diretto(
	bStart:=  , 
	nAddr:= , 
	eAddrType:=, 
	eCommandPriority:= , 
	nArcPowerLevel:= , 
	bBusy=> , 
	bError=> , 
	nErrorId=> , 
	stCommandBuffer:= DALI_BUFFER2);

END_PROGRAM

// ---- POUs/ProjetcFB/Luci_Mov_Dali.TcPOU
FUNCTION_BLOCK Luci_Mov_Dali
VAR_INPUT
	Movimento:BOOL;
	Delay:TIME;
	Addr:BYTE;
	Lux:WORD;
END_VAR
VAR_OUTPUT
END_VAR
VAR
	Tempo_oFF: TOF;
	mempower: WORD;
	Luce: FB_DALIV2DirectArcPowerControl;
	power:BYTE;
	TRx:BOOL;
	timer:WORD;
END_VAR

timer:=Timer+1;
Tempo_oFF(IN:=Movimento , PT:=Delay , Q=> , ET=> );
IF Tempo_off.Q THEN 
	power:=254;
ELSE
	power:=0;
END_IF
IF power=0 AND lux>30 AND timer=25000 THEN
	TRx:=TRUE;
ELSIF power <> mempower THEN
	TRx:=TRUE;
	mempower:=power;
ELSE
	TRx:=FALSE;
END_IF
Luce(
	bStart:=TRx  , 
	nAddr:=ADDR, 
	eAddrType:= 0, 
	eCommandPriority:= , 
	nArcPowerLevel:=power , 
	bBusy=> , 
	bError=> , 
	nErrorId=> , 
	stCommandBuffer:=DALI_BUFFER2 );
	
IF timer>25000 THEN
	timer:=0;
END_IF

END_FUNCTION_BLOCK

// ---- POUs/Ekey.TcPOU
PROGRAM Ekey
VAR
	ekey_comm: FB_EKEY_Communication;
	ekey_in AT %I*: kl6indata22b;
	ekey_out AT %Q*: kl6outdata22b;
	ekey_buffer: ST_EKEY_CommandBuffer;
	template_utenti: ST_EKEY_FingerTemplate;
END_VAR

// Comunicazione Ekey	
ekey_comm(
	bEnable:= TRUE, 
	eMode:= seriallinemode_kl6_22b_standard, 
	pComIn:= ADR(ekey_in), 
	pComOut:= ADR(ekey_out), 
	uiSizeComIn:= SIZEOF(ekey_in), 
	bBusy=> , 
	bError=> , 
	udiErrorID=> , 
	stCommandBuffer:= ekey_buffer);
//Scanner Ekey cancello carraio
ekey_scanner_cancello(
	bEnable:= TRUE, 
	sSN:= '31160073', 
	bNewFinger:= , 
	byFingerID:= , 
	byUserID:= , 
	bFingerControlRelay:= , 
	eEnrollmentFunction:= eEKEYEnrollNormal, 
	bRemoveUser:= , 
	bRemoveAllUsers:= , 
	byRemoveUserID:= , 
	eLedFunction:= , 
	diLedClock:= , 
	bRelayOn:= , 
	bResetAll:= , 
	bReadTemplate:= , 
	bWriteUser:= , 
	bWriteTemplate:= , 
	byReadTempFingerID:= , 
	byReadTempUserID:= , 
	bySetUserID:= , 
	byWriteTempFingerID:= , 
	byWriteTempUserID:= , 
	stWriteTemplate:= , 
	bNewRFID:= , 
	bReadRFID:= , 
	bWriteRFID:= , 
	bSwitchFSensor_ON:= , 
	bSwitchFSensor_OFF:= , 
	bRFIDControlRelay:= , 
	byRFIDUserID:= , 
	arrWriteRFID:= , 
	bBusy=> , 
	bError=> , 
	udiErrorID=> , 
	bBufferOverload=> , 
	eState=> , 
	bReceived=> , 
	byRecUserID=> , 
	byRecFingerID=> , 
	byRecTempUserID=> , 
	byRecTempFingerID=> , 
	byRecRFIDUserID=> , 
	bBadFinger=> , 
	dwBadFingers=> , 
	bGoodFinger=> , 
	dwMaxConfigUser=> , 
	dwMaxConfigFinger=> , 
	stRecTemplate=> template_utenti, 
	arrRecRFID=> , 
	stCommandBuffer:= ekey_buffer);
	
//Scanner Ekey produzione
ekey_scanner_produzione(
	bEnable:= TRUE, 
	sSN:= '24180820', 
	bNewFinger:= , 
	byFingerID:= , 
	byUserID:= , 
	bFingerControlRelay:= , 
	eEnrollmentFunction:= eEKEYEnrollNormal, 
	bRemoveUser:= , 
	bRemoveAllUsers:= , 
	byRemoveUserID:= , 
	eLedFunction:= , 
	diLedClock:= , 
	bRelayOn:= , 
	bResetAll:= , 
	bReadTemplate:= , 
	bWriteUser:= , 
	bWriteTemplate:= , 
	byReadTempFingerID:= , 
	byReadTempUserID:= , 
	bySetUserID:= , 
	byWriteTempFingerID:= , 
	byWriteTempUserID:= , 
	stWriteTemplate:= , 
	bNewRFID:= , 
	bReadRFID:= , 
	bWriteRFID:= , 
	bSwitchFSensor_ON:= , 
	bSwitchFSensor_OFF:= , 
	bRFIDControlRelay:= , 
	byRFIDUserID:= , 
	arrWriteRFID:= , 
	bBusy=> , 
	bError=> , 
	udiErrorID=> , 
	bBufferOverload=> , 
	eState=> , 
	bReceived=> , 
	byRecUserID=> , 
	byRecFingerID=> , 
	byRecTempUserID=> , 
	byRecTempFingerID=> , 
	byRecRFIDUserID=> , 
	bBadFinger=> , 
	dwBadFingers=> , 
	bGoodFinger=> , 
	dwMaxConfigUser=> , 
	dwMaxConfigFinger=> , 
	stRecTemplate=> , 
	arrRecRFID=> , 
	stCommandBuffer:= ekey_buffer);
	
//Scanner Ekey porta ingresso
ekey_scanner_ingresso(
	bEnable:= TRUE, 
	sSN:= '37160694', 
	bNewFinger:= , 
	byFingerID:= , 
	byUserID:= , 
	bFingerControlRelay:= , 
	eEnrollmentFunction:= eEKEYEnrollNormal, 
	bRemoveUser:= , 
	bRemoveAllUsers:= , 
	byRemoveUserID:= , 
	eLedFunction:= , 
	diLedClock:= , 
	bRelayOn:= , 
	bResetAll:= , 
	bReadTemplate:= , 
	bWriteUser:= , 
	bWriteTemplate:= , 
	byReadTempFingerID:= , 
	byReadTempUserID:= , 
	bySetUserID:= , 
	byWriteTempFingerID:= , 
	byWriteTempUserID:= , 
	stWriteTemplate:= template_utenti, 
	bNewRFID:= , 
	bReadRFID:= , 
	bWriteRFID:= , 
	bSwitchFSensor_ON:= , 
	bSwitchFSensor_OFF:= , 
	bRFIDControlRelay:= , 
	byRFIDUserID:= , 
	arrWriteRFID:= , 
	bBusy=> , 
	bError=> , 
	udiErrorID=> , 
	bBufferOverload=> , 
	eState=> , 
	bReceived=> , 
	byRecUserID=> , 
	byRecFingerID=> , 
	byRecTempUserID=> , 
	byRecTempFingerID=> , 
	byRecRFIDUserID=> , 
	bBadFinger=> , 
	dwBadFingers=> , 
	bGoodFinger=> , 
	dwMaxConfigUser=> , 
	dwMaxConfigFinger=> , 
	stRecTemplate=> , 
	arrRecRFID=> , 
	stCommandBuffer:= ekey_buffer);
	
ekey_scanner_cancello.arrWriteRFID:=ekey_scanner_produzione.arrRecRFID;
//Registrazione del dito dell'utente
IF hmi_finger THEN
	ekey_scanner_produzione.byUserID:=ekey_scanner_produzione.byRecUserID;
	ekey_Scanner_produzione.byFingerID:=1(*ekey_Scanner_produzione.byRecFingerID*);
	IF ekey_scanner_produzione.bGoodFinger THEN
		ekey_scanner_produzione.bNewFinger:=TRUE;
	ELSE
		ekey_scanner_produzione.bNewFinger:=FALSE;
	END_IF
END_IF
//Registrazione del RFID dell'utente
IF hmi_finger_RFID THEN
	ekey_scanner_produzione.byRFIDUserID:=HMI_userRFID;
	ekey_scanner_produzione.bNewRFID:=TRUE;
ELSE
	ekey_scanner_produzione.bNewRFID:=FALSE;
END_IF

END_PROGRAM

// ---- POUs/Riscaldamento.TcPOU
PROGRAM Riscaldamento
VAR
	Sabiana1: Speed_Sabiana;
	Sabiana2: Speed_Sabiana;
	Sabiana3: Speed_Sabiana;
	Sabiana4: Speed_Sabiana;
	Sabiana5: Speed_Sabiana;
	Sabiana6: Speed_Sabiana;
	Temp_Prod1: DALI_TK_SR07_rh;
	areotermi AT %Q*: ARRAY [1..10] OF areotermo;
	night:BOOL;
	richiesta_caldaia AT %Q*: BOOL;
	pompa_prod1 AT %Q*: BOOL;
	pompa_prod2 AT %Q*: BOOL;
	f_coil1: F_COIL;
	f_coil2: F_COIL;
	f_coil3: F_COIL;
	f_coil4: F_COIL;
	f_coil5: F_COIL;
	f_coil6: F_COIL;
	f_coil7: F_COIL;
	f_coil8: F_COIL;
	f_coil9: F_COIL;
	f_coil10: F_COIL;
	delay_onciller: TON;
	CILLER_ON: BOOL;
	temp_ciller AT %I*: INT;
	run_pompaprod AT %I*: BOOL;
	switch_pompa_prod: INT;
	forza_inverno_misto: BOOL;
	riscaldamento_man: BOOL:=FALSE;
	forza_aer_uffici: BOOL;
	forza_richiesta_caldaia: BOOL;
	forza_pompa_prod1: BOOL;
	forza_pompa_prod2: BOOL;
	forza_Sabiana1L: BOOL;
	forza_Sabiana1H: BOOL;
	forza_Sabiana2L: BOOL;
	forza_Sabiana2H: BOOL;
	forza_Sabiana3L: BOOL;
	forza_Sabiana3H: BOOL;
	forza_Sabiana4L: BOOL;
	forza_Sabiana4H: BOOL;
	forza_Sabiana5L: BOOL;
	forza_Sabiana5H: BOOL;
	forza_Sabiana6L: BOOL;
	forza_Sabiana6H: BOOL;
	sab1_state: INT;
END_VAR

//Temperature Capannone
Temp_Prod1(ID:= 16#019E5ACD, Temp=> TEMPz0, Umidity=> HMI_umidita);
IF NOT Sabiana1L AND NOT Sabiana1H THEN
	sab1_state:=0;
ELSIF Sabiana1L AND NOT Sabiana1H THEN
	sab1_state:=1;
ELSIF NOT Sabiana1L AND Sabiana1H THEN
	sab1_state:=2;
END_IF
IF riscaldamento_man THEN //Modalità MANUALE
	aer_uffici:=forza_aer_uffici;
	richiesta_caldaia:=forza_richiesta_caldaia;
	switch_pompa_prod:=2;
	pompa_prod1:=forza_pompa_prod1;
	pompa_prod2:=forza_pompa_prod2;
	Sabiana1L:=forza_Sabiana1L;
	Sabiana1H:=forza_Sabiana1H;
	Sabiana2L:=forza_Sabiana2L;
	Sabiana2H:=forza_Sabiana2H;
	Sabiana3L:=forza_Sabiana3L;
	Sabiana3H:=forza_Sabiana3H;
	Sabiana4L:=forza_Sabiana4L;
	Sabiana4H:=forza_Sabiana4H;
	Sabiana5L:=forza_Sabiana5L;
	Sabiana5H:=forza_Sabiana5H;
	Sabiana6L:=forza_Sabiana6L;
	Sabiana6H:=forza_Sabiana6H;

ELSE //Modalità AUTOMATICO
(* Areazione *)
aer_uffici:=allarme_Attivo=0 (*NOT Allarme*);

//Gestione Pompa Caldaia
richiesta_caldaia:=	sabiana1.pompa OR
					sabiana2.pompa OR
					sabiana3.pompa OR
					sabiana4.pompa OR
					sabiana5.pompa OR
					sabiana6.pompa OR
					temp_ciller < 600 OR
					f_coil1.C2_pompa OR
					f_coil2.C2_pompa OR
					f_coil3.C2_pompa OR
					f_coil4.C2_pompa OR
					f_coil5.C2_pompa OR
					f_coil6.C2_pompa OR
					f_coil7.C2_pompa OR
					f_coil8.C2_pompa OR
					f_coil9.C2_pompa OR
					f_coil10.C2_pompa ;
				
switch_pompa_prod:=ora_plc.TIMESTR.wDay MOD 2;

//Switch tra le due pompe in funzione del giorno pari o dispari
IF switch_pompa_prod=0 THEN
	pompa_prod1:=run_pompaprod ;
	pompa_prod2:=FALSE;
ELSIF switch_pompa_prod=1 THEN
	pompa_prod2:=run_pompaprod;
	pompa_prod1:=FALSE;
END_IF;

(*Gestione Sabiana*)
	Sabiana1(
		modo:= HMI_SabianaManCTRL[1], 
		Hmodo:= HeatingdMode , 
		Tzona:= tempz0, 
		Trif:= ,//hmi_tempprod, 
		Hspeed:= , 
		Tciller:= temp_ciller,
		ToffCiller:=TempOffSabiana1,  
		TH20:=(*Th20_CaldaiaOK*) run_pompaprod OR night,
		L=> Sabiana1L, 
		H=> Sabiana1H,
		Pompa=>);
	Sabiana2(
		modo:= HMI_SabianaManCTRL[2], 
		Hmodo:= HeatingdMode , 
		Tzona:= tempz0, 
		Trif:= ,//hmi_tempprod, 
		Hspeed:= , 
		Tciller:= temp_ciller,
		ToffCiller:=TempOffSabiana2 ,
		TH20:=(*Th20_CaldaiaOK*) run_pompaprod OR night,
		L=> Sabiana2L, 
		H=> Sabiana2H,
		Pompa=>);
	Sabiana3(
		modo:= HMI_SabianaManCTRL[3], 
		Hmodo:= HeatingdMode , 
		Tzona:= tempz0, 
		Trif:= ,//hmi_tempprod, 
		Hspeed:= , 
		Tciller:= temp_ciller,
		ToffCiller:=TempOffSabiana3 ,
		TH20:=(*Th20_CaldaiaOK*) run_pompaprod OR night,
		L=> Sabiana3L, 
		H=> Sabiana3H,
		Pompa=>);
	Sabiana4(
		modo:= HMI_SabianaManCTRL[4], 
		Hmodo:= HeatingdMode , 
		Tzona:= tempz0, 
		Trif:= ,//hmi_tempprod, 
		Hspeed:= , 
		Tciller:= temp_ciller,
		ToffCiller:=TempOffSabiana4 ,
		TH20:=(*Th20_CaldaiaOK*) run_pompaprod OR night,
		L=> Sabiana4L, 
		H=> Sabiana4H,
		Pompa=>);
	Sabiana5(
		modo:= HMI_SabianaManCTRL[5], 
		Hmodo:= HeatingdMode , 
		Tzona:= tempz0, 
		Trif:= ,//hmi_tempprod, 
		Hspeed:= , 
		Tciller:= temp_ciller,
		ToffCiller:=TempOffSabiana5 ,
		TH20:=(*Th20_CaldaiaOK*) run_pompaprod OR night,
		L=> Sabiana5L, 
		H=> Sabiana5H,
		Pompa=>);
	Sabiana6(
		modo:= HMI_SabianaManCTRL[6], 
		Hmodo:= HeatingdMode , 
		Tzona:= tempz0, 
		Trif:= ,//hmi_tempprod, 
		Hspeed:= , 
		Tciller:= temp_ciller,
		ToffCiller:=TempOffSabiana6 ,
		TH20:=(*Th20_CaldaiaOK*) run_pompaprod OR night,
		L=> Sabiana6L, 
		H=> Sabiana6H,
		Pompa=>);
		
//UFFICI
//GESTIONE ESTATE INVERNO
OUT_CILLER_ESTATE:=OFFICE_VHAC_EI;
//GESTIONE MODO CILLER
IF 		OUT_CILLER_ESTATE THEN
		OFFICE_vhac_MODE:=0; // 0 ESTATE 
ELSIF 	NOT OUT_CILLER_ESTATE AND (Temp_OUTSIDE<-1 OR forza_inverno_misto) THEN
		OFFICE_vhac_MODE:=2; // 2 INVERNO MISTO 
ELSIF 	NOT OUT_CILLER_ESTATE  THEN
		OFFICE_vhac_MODE:=1; // 1 INVERNO PDC
END_IF

(*Gestione Pompa Ciller*)
delay_onciller(IN:=ciller_on , PT:= T#5M, Q=>OUT_CILLER_ON , ET=> );
CILLER_ON:= 
	f_coil1.C1_pompa OR
	f_coil2.C1_pompa OR
	f_coil3.C1_pompa OR
	f_coil4.C1_pompa OR
	f_coil5.C1_pompa OR
	f_coil6.C1_pompa OR
	f_coil7.C1_pompa OR
	f_coil8.C1_pompa OR
	f_coil9.C1_pompa OR
	f_coil10.C1_pompa OR
	Temp_OUTSIDE<-2 ;
//Ingresso
f_coil1(
	C1_TH2o:= th20_pompacaloreok, 
	C2_TH2o:= TRUE, 
	mode:= OFFICE_vhac_MODE, 
	T_AMB:= Tempz1,//-HMI_var_tempuff[1]), 
	T_RIF:= ,//HMI_TEMPuff[1], 
	winterON:=INT_TO_BOOL(cononz1),
	Forza_VOpen:= ciller_on, 
	C1_VOPEN=>areotermi[1].VHL1, 
	C2_VOPEN=>areotermi[1].VHL2, 
	V1=>areotermi[1].Speed1, 
	V2=>areotermi[1].Speed2, 
	V3=>areotermi[1].Speed3, 
	C1_pompa=> , 
	C2_Pompa=> );	
//Amministrazione
f_coil2(
	C1_TH2o:= th20_pompacaloreok, 
	C2_TH2o:= TRUE, 
	mode:= OFFICE_vhac_MODE, 
	T_AMB:= Tempz3,//-HMI_var_tempuff[2]), 
	T_RIF:= ,//HMI_TEMPuff[2], 
	winterON:= INT_TO_BOOL (cononz2),
	Forza_VOpen:= ciller_on, 
	C1_VOPEN=> areotermi[2].VHL1, 
	C2_VOPEN=> areotermi[2].VHL2, 
	V1=> areotermi[2].Speed1, 
	V2=> areotermi[2].Speed2, 
	V3=> areotermi[2].Speed3, 
	C1_pompa=> , 
	C2_Pompa=> );
//Direzione
f_coil3(
	C1_TH2o:= th20_pompacaloreok, 
	C2_TH2o:= TRUE, 
	mode:= OFFICE_vhac_MODE, 
	T_AMB:= Tempz3,//-HMI_var_tempuff[3]), 
	T_RIF:= ,//HMI_TEMPuff[3], 
	winterON:= INT_TO_BOOL(cononz3),
	Forza_VOpen:= CILLER_ON, 
	C1_VOPEN=> areotermi[3].VHL1, 
	C2_VOPEN=> areotermi[3].VHL2, 
	V1=> areotermi[3].Speed1, 
	V2=> areotermi[3].Speed2, 
	V3=> areotermi[3].Speed3, 
	C1_pompa=> , 
	C2_Pompa=> );
//Sala Riunioni
f_coil4(
	C1_TH2o:= th20_pompacaloreok, 
	C2_TH2o:= TRUE, 
	mode:= OFFICE_vhac_MODE, 
	T_AMB:= tempz4,//-HMI_var_tempuff[4]), 
	T_RIF:= ,//HMI_TEMPuff[4], 
	winterON:= INT_TO_BOOL(cononz4) OR meetingroom_active,
	Forza_VOpen:= CILLER_ON , 
	C1_VOPEN=> areotermi[4].VHL1, 
	C2_VOPEN=> areotermi[4].VHL2, 
	V1=> areotermi[4].Speed1, 
	V2=> areotermi[4].Speed2, 
	V3=> areotermi[4].Speed3, 
	C1_pompa=> , 
	C2_Pompa=> );
f_coil5(
	C1_TH2o:= th20_pompacaloreok, 
	C2_TH2o:= TRUE, 
	mode:= OFFICE_vhac_MODE, 
	T_AMB:= tempz4,//-HMI_var_tempuff[4]), 
	T_RIF:= ,//HMI_TEMPuff[4], 
	winterON:= INT_TO_BOOL(cononz4) OR meetingroom_active,
	Forza_VOpen:= CILLER_ON, 
	C1_VOPEN=> areotermi[5].VHL1, 
	C2_VOPEN=> areotermi[5].VHL2, 
	V1=> areotermi[5].Speed1, 
	V2=> areotermi[5].Speed2, 
	V3=>areotermi[5].Speed3, 
	C1_pompa=> , 
	C2_Pompa=> );
//Ufficio Tecnico
f_coil6(
	C1_TH2o:= th20_pompacaloreok, 
	C2_TH2o:= TRUE, 
	mode:= OFFICE_vhac_MODE, 
	T_AMB:= tempz5,//-HMI_var_tempuff[5]), 
	T_RIF:= ,//HMI_TEMPuff[5], 
	winterON:= INT_TO_BOOL(cononz5),
	Forza_VOpen:= CILLER_ON, 
	C1_VOPEN=> areotermi[6].VHL1, 
	C2_VOPEN=> areotermi[6].VHL2, 
	V1=> areotermi[6].Speed1, 
	V2=> areotermi[6].Speed2, 
	V3=>areotermi[6].Speed3, 
	C1_pompa=> , 
	C2_Pompa=> );
f_coil7(
	C1_TH2o:= th20_pompacaloreok, 
	C2_TH2o:= TRUE, 
	mode:= OFFICE_vhac_MODE, 
	T_AMB:= tempz5,//-HMI_var_tempuff[5]), 
	T_RIF:= ,//HMI_TEMPuff[5], 
	winterON:= INT_TO_BOOL(cononz5),
	Forza_VOpen:= CILLER_ON , 
	C1_VOPEN=> areotermi[7].VHL1, 
	C2_VOPEN=> areotermi[7].VHL2, 
	V1=> areotermi[7].Speed1, 
	V2=> areotermi[7].Speed2, 
	V3=> areotermi[7].Speed3, 
	C1_pompa=> , 
	C2_Pompa=> );
//Ufficio Produzione
f_coil8(
	C1_TH2o:= th20_pompacaloreok, 
	C2_TH2o:= TRUE, 
	mode:= OFFICE_vhac_MODE, 
	T_AMB:= tempz6,//-HMI_var_tempuff[6]),
	T_RIF:= ,//HMI_TEMPuff[5], 
	winterON:= INT_TO_BOOL(cononz6),
	Forza_VOpen:= CILLER_ON , 
	C1_VOPEN=> areotermi[8].VHL1, 
	C2_VOPEN=> areotermi[8].VHL2, 
	V1=> areotermi[8].Speed1, 
	V2=> areotermi[8].Speed2, 
	V3=> areotermi[8].Speed3, 
	C1_pompa=> , 
	C2_Pompa=> );
f_coil9(
	C1_TH2o:= th20_pompacaloreok, 
	C2_TH2o:= TRUE, 
	mode:= OFFICE_vhac_MODE, 
	T_AMB:= tempz6,//-HMI_var_tempuff[6]), 
	T_RIF:= ,//HMI_TEMPuff[5],
	winterON:= INT_TO_BOOL(cononz6), 
	Forza_VOpen:= CILLER_ON , 
	C1_VOPEN=> areotermi[9].VHL1, 
	C2_VOPEN=> areotermi[9].VHL2, 
	V1=> areotermi[9].Speed1, 
	V2=> areotermi[9].Speed2, 
	V3=> areotermi[9].Speed3, 
	C1_pompa=> , 
	C2_Pompa=> );
//Locale Svago
f_coil10(
	C1_TH2o:= th20_pompacaloreok, 
	C2_TH2o:= TRUE, 
	mode:= OFFICE_vhac_MODE, 
	T_AMB:= tempz7, 
	T_RIF:= ,//HMI_TEMPuff[7], 	
	winterON:= INT_TO_BOOL(cononz7),
	Forza_VOpen:= ciller_on, 
	C1_VOPEN=> areotermi[10].VHL1, 
	C2_VOPEN=> areotermi[10].VHL2, 
	V1=> areotermi[10].Speed1, 
	V2=> areotermi[10].Speed2, 
	V3=> areotermi[10].Speed3, 
	C1_pompa=> , 
	C2_Pompa=> );
	(*IF NOT OFFICE_VHAC_EI THEN
		IF 1230<=time_now AND time_now<=1330 THEN
			f_coil10.T_AMB:= (tempz7-HMI_var_tempuff[7]);
		ELSE
			f_coil10.T_AMB:=tempz7;
		END_IF
	ELSE
		f_coil10.T_AMB:=tempz7;
	END_IF*)
IF OFFICE_VHAC_EI THEN //Se estate ON
	//HMI_TEMPuff:=280;
END_IF

IF NOT OFFICE_VHAC_EI THEN (*Se è inverno*)
	IF ORA_PLC.TIMESTR.wHour>=6 AND ORA_PLC.TIMESTR.wHour<=17 THEN
		//hmi_tempprod:=160;
		//HMI_TEMPuff:=240;
		night:=FALSE;
		sabiana1.Trif:=hmi_tempprod;
		sabiana2.Trif:=hmi_tempprod;
		sabiana3.Trif:=hmi_tempprod;
		sabiana4.Trif:=hmi_tempprod;
		sabiana5.Trif:=hmi_tempprod;
		sabiana6.Trif:=hmi_tempprod;
		f_coil1.T_RIF:=HMI_tempuff[1];
		f_coil2.T_RIF:=HMI_tempuff[2];
		f_Coil3.T_RIF:=HMI_tempuff[3];
		f_coil4.T_RIF:=HMI_tempuff[4];
		f_coil5.T_RIF:=HMI_tempuff[4];
		f_coil6.T_RIF:=HMI_tempuff[5];
		f_coil7.T_RIF:=HMI_tempuff[5];
		f_coil8.T_RIF:=HMI_tempuff[5];
		f_coil9.T_RIF:=HMI_tempuff[5];
		f_Coil10.T_RIF:=HMI_tempuff[7];
	ELSE
		night:=TRUE;
		sabiana1.Trif:=140;
		sabiana2.Trif:=140;
		sabiana3.Trif:=140;
		sabiana4.Trif:=140;
		sabiana5.Trif:=140;
		sabiana6.Trif:=140;
		f_coil1.T_RIF:=160;
		f_coil2.T_RIF:=160;
		f_coil3.T_RIF:=160;
		f_coil4.T_RIF:=160;
		f_coil5.T_RIF:=160;
		f_coil6.T_RIF:=160;
		f_coil7.T_RIF:=160;
		f_coil8.T_RIF:=160;
		f_coil9.T_RIF:=160;
		f_coil10.T_RIF:=160;
	END_IF
END_IF
END_IF

END_PROGRAM

// ---- POUs/ProjetcFB/Speed_Sabiana.TcPOU
FUNCTION_BLOCK Speed_Sabiana
VAR_INPUT
	modo : BYTE;(*Tipo Velocità*)
	Hmodo: BYTE ;(*tipo riscaldamento*)
	Tzona: UINT; (*Temperatura attuale della zona*)
	Trif:UINT;	(*temperatura di riferimento programmata*)
	Hspeed:BOOL; (*per forzare veloctà alta*)
	TH20:BOOL;
	TCiller:INT;
	TCiller1:BOOL;
	Toffciller:INT;
END_VAR
VAR_OUTPUT
	L :BOOL;
	H :BOOL;
	pompa:BOOL;
END_VAR
VAR
END_VAR

	(*--Sabiana X --*)
	//TCiller1:=Toffciller-Tciller(*Tciller/10*);
	IF Tciller>(Toffciller+1) THEN
		tciller1:=TRUE;
	ELSIF tciller<toffciller THEN
		tciller1:=FALSE;
	END_IF
	IF 	Hmodo=0 THEN
			L :=FALSE;
			H :=FALSE;
			pompa:=FALSE;
	ELSIF Hmodo=1 THEN
		pompa:=TRUE;
		IF modo=1 THEN
			L :=TRUE;
			H :=FALSE;
		ELSIF modo=2 THEN
			L :=FALSE;
			H :=TRUE;
		ELSE
			L :=FALSE;
			H :=FALSE;
		END_IF;
	ELSIF Hmodo=2 THEN
		IF tzona<Trif AND NOT Hspeed AND tciller1(*>Toffciller*) THEN
			L :=TRUE AND TH20;
			H :=FALSE;
			pompa:=TRUE;
		ELSIF tzona<Trif AND Hspeed AND Tciller1(*>Toffciller*) THEN
			L :=FALSE;
			H :=TRUE AND TH20;
			pompa:=TRUE;
		ELSIF tzona>=Trif OR Tciller<=Toffciller THEN
			L :=FALSE;
			H :=FALSE;
			pompa:=FALSE;
		END_IF
	ELSIF Hmodo=3 THEN
		IF prod_summer_fan=0 THEN
			L :=FALSE;
			H :=FALSE;
			pompa:=FALSE;
		ELSIF prod_summer_fan=1 THEN
			L :=TRUE;
			H :=FALSE;
			pompa:=FALSE;
		ELSIF prod_summer_fan=2 THEN
			L :=FALSE;
			H :=TRUE;
			pompa:=FALSE;
		END_IF
	END_IF

END_FUNCTION_BLOCK

// ---- POUs/ProjetcFB/DALI_TK_SR07_rh.TcPOU
FUNCTION_BLOCK DALI_TK_SR07_rh
VAR_INPUT
	ID: DWORD;
END_VAR
VAR_OUTPUT
	Temp : UINT; //Valore * 10 - 10,0°C => 100
	Umidity :BYTE; //Valore in %
END_VAR
VAR
	READ: FB_Rec_Generic;
	temperatura: DINT;
	umidita: DINT;
END_VAR

READ(
	str_KL6581:=enocean_buffer , 
	byNode:=1 , 
	dw_ID:=ID , 
	ar_Value=> , 
	by_Node=> , 
	by_STATE=> , 
	bReceive=> , 
	EnOceanTyp=> );
temperatura:=TRUNC(read.ar_Value[1]/0.625);	
temp:=DINT_TO_UINT (temperatura);
umidita:=TRUNC(read.ar_Value[2]/2.5);
Umidity:=DINT_TO_byte (umidita);

END_FUNCTION_BLOCK

// ---- POUs/ProjetcFB/F_COIL.TcPOU
FUNCTION_BLOCK F_COIL
VAR_INPUT
	C1_TH2o:BOOL;
	C2_TH2o:BOOL;
	mode:BYTE; // 0= ESTATE - 1 INVERNO PDC - 2 INVERNO MISTO 
	T_AMB:UINT;
	T_RIF:UINT;
	Forza_VOpen:BOOL;
	winterON: BOOL;
END_VAR
VAR_OUTPUT
	C1_VOPEN:BOOL;
	C2_VOPEN:BOOL;
	V1:BOOL;
	V2:BOOL;
	V3:BOOL;
	C1_pompa:BOOL;
	C2_Pompa:BOOL;
END_VAR
VAR
END_VAR

IF T_amb>T_rif AND mode=0 AND winterON THEN
	C1_VOPEN:=TRUE;
	C2_VOPEN:=FALSE;
	C1_pompa:=TRUE;
	C2_Pompa:=FALSE;
ELSIF (T_amb<=T_rif OR NOT winterON) AND mode=0  THEN
	C1_VOPEN:=FALSE;
	C2_VOPEN:=FALSE;
	C1_pompa:=FALSE;
	C2_Pompa:=FALSE;
ELSIF T_amb<T_rif AND mode=1 THEN
	C1_VOPEN:=TRUE;
	C2_VOPEN:=FALSE;
	C1_pompa:=TRUE;
	C2_Pompa:=FALSE;
ELSIF T_amb<T_rif AND mode=2 THEN
	C1_VOPEN:=TRUE;
	C2_VOPEN:=TRUE;
	C1_pompa:=TRUE;
	C2_Pompa:=TRUE;
ELSIF T_amb>=T_rif AND (MODE=1 OR MODE=2) THEN
	C1_VOPEN:=FALSE;
	C2_VOPEN:=FALSE;
	C1_pompa:=FALSE;
	C2_Pompa:=FALSE;
END_IF
IF Forza_VOpen THEN
	C1_VOPEN:=TRUE;
END_IF
IF MODE=0 AND T_AMB>T_RIF AND winteron THEN
	V1:=FALSE;
	V2:=TRUE;
	V3:=FALSE;
ELSIF MODE=0 AND (T_AMB<=T_RIF OR NOT winterON) THEN
	V1:=FALSE;
	V2:=FALSE;
	V3:=FALSE;	
ELSIF  T_amb>(T_rif-5)AND T_amb<T_rif THEN 
	V1:=TRUE;
	V2:=FALSE;
	V3:=FALSE;
ELSIF (T_amb>(T_rif-10) AND T_amb<T_rif) OR ( T_amb<T_rif AND NOT c1_th2o) THEN 
	V1:=FALSE;
	V2:=TRUE;
	V3:=FALSE;
ELSIF  T_amb<T_rif AND c1_th2o THEN 
	V1:=FALSE;
	V2:=FALSE;
	V3:=TRUE;
ELSE
	V1:=FALSE;
	V2:=FALSE;
	V3:=FALSE;
END_IF

END_FUNCTION_BLOCK

// ---- POUs/LUCI.TcPOU
PROGRAM LUCI
VAR
	luci_esterne AT %Q*:BOOL;
	lux_capannone: EnO_TK_SR65_LI;
	luci_DIREZIONE: Dali_arcpower_control;
	luci_riunioni: Dali_arcpower_control;
	luci_capannone: Dali_arcpower_control;
	HMI_ctrl_luci: INT; //Variabile per gestione Linear Gauge luci capannone
	movimento_server: EnO_TK_SR_MDS_BAT;
	luce_server: Dali_arcpower_control;
	delay_luce_server: TOF;
	Ulux_0: ULUX_STD;
	ulux_1: ULUX_STD;
	ulux_2: ULUX_STD;
	Ulux_3: ULUX_STD;
	ulux_4: ULUX_STD;
	ulux_5: ULUX_STD;
	ulux_6: ULUX_STD;
	luce_17: Dali_arcpower_control;
	luce_18: Dali_arcpower_control;
	luce_19: Dali_arcpower_control;
	luce_20: Dali_arcpower_control;
	group_0: Dali_arcpower_control;
	group_1: Dali_arcpower_control;
	group_2: Dali_arcpower_control;
	group_3: Dali_arcpower_control;
	group_5: Dali_arcpower_control;
	group_6: Dali_arcpower_control;
	group_7: Dali_arcpower_control;
	group_8: Dali_arcpower_control;
	group_9: Dali_arcpower_control;
	group_10: Dali_arcpower_control;
	On_Off_luce1: Comando_LuceDali;
	luce_1: Dali_arcpower_control;
	On_Off_Gruppo0: Comando_LuceDali;
	gruppo0: Dali_arcpower_control;
	LUXEXTREF: BYTE:=20;
	ins_AUTOluce_capannone: F_TRIG;
	luci_ON_auto: BOOL; //Accensione luce amministrazione senza allarme
END_VAR

//03 LUCI

//03.01 Luci Capannone
	lux_capannone(ID:=16#01A465FE , LUX=> , status=> ,);
		//Accensione_luci(CLK:=allarme , Q=>light_on );
		//Spegnimento_luci(CLK:=allarme, Q=>light_off);
	ins_AUTOluce_capannone(CLK:=time_now=0730 , Q=> );
	IF ins_AUTOluce_capannone.Q THEN
		luci_capannone_aut:=TRUE;
	END_IF
	IF allarme_Attivo<>0 THEN
		luci_capannone.light_level:=0;
	ELSIF allarme_Attivo=0 AND (time_now<0655 OR time_now>1705 OR (time_now<1325 AND time_now>1235)) AND luci_capannone_aut THEN
		luci_capannone.light_level:=150;	
	ELSE 
		luci_capannone.light_level:=HMI_luci_capannone;
	END_IF
	luci_capannone(light_level:= , ADDR:= , MODE:=2 , daliBuffer:=DALI_BUFFER1 );

//03.02 Luci esterne
	IF	(LUX_OUTSIDEF<LUXEXTREF OR LUX_OUTSIDER<LUXEXTREF OR LUX_OUTSIDEL<LUXEXTREF) OR HMI_luce_3 THEN
		luci_esterne:=TRUE;
	ELSE
		luci_esterne:=FALSE;
	END_IF
	luce3:=luci_esterne;
//03.03 LUCI UFFICIO
	//Generale Uffici
	IF allarme_Attivo<>0 THEN
		luci_ufficio_off:=TRUE;
		luci_ON_auto:=FALSE;
	ELSE
		luci_ufficio_off:=FALSE;
		luci_ON_auto:=TRUE;
	END_IF
		
//Ingresso (gruppi:0 e 1) ID:0
	ulux_0(
		ID:= 0, 
		luci_OFF:= luci_ufficio_off OR HMI_luci_off[0], 
		luci_ON:= HMI_luci_on[0], 
		time_delay:= , 
		condiz_ON_OFF:= HMI_cond[0],
		arc_level=> , 
		temp=> Tempz1, 
		funzione_1=> , 
		moviment_active=> , 
		condiz=> cononz1);
	group_0(light_level:= ulux_0.arc_level, ADDR:= 0, MODE:= 1, daliBuffer:= DALI_BUFFER2);
	group_1(light_level:= ulux_0.arc_level, ADDR:= 1, MODE:= 1, daliBuffer:= DALI_BUFFER2);
//Amministrazione Gruppo:2 ID:1
	ulux_1(
		ID:= 1, 
		luci_OFF:= luci_ufficio_off OR HMI_luci_off[1], 
		luci_ON:= HMI_luci_on[1], //OR luci_ON_auto, 
		time_delay:= , 
		condiz_ON_OFF:= HMI_cond[1],
		arc_level=> , 
		temp=> Tempz2, 
		funzione_1=> , 
		moviment_active=> , 
		condiz=> cononz2);
	group_2(light_level:= ulux_1.arc_level, ADDR:= 2, MODE:= 1, daliBuffer:= DALI_BUFFER2);
//Direzione Gruppo:3 ID:2
	ulux_2(
		ID:= 2, 
		luci_OFF:= luci_ufficio_off OR HMI_luci_off[2], 
		luci_ON:= HMI_luci_on[2], 
		time_delay:= , 
		condiz_ON_OFF:= HMI_cond[2],
		arc_level=> , 
		temp=> Tempz3, 
		funzione_1=> , 
		moviment_active=> , 
		condiz=> cononz3);
	group_3(light_level:= ulux_2.arc_level, ADDR:= 3, MODE:= 1, daliBuffer:= DALI_BUFFER2);
//Sala riunioni Gruppo:4 ID:3
	ulux_3(
		ID:= 3, 
		luci_OFF:= luci_ufficio_off, //OR HMI_luci_off[3], 
		luci_ON:= ,//HMI_luci_on[3], 
		time_delay:= T#10M, 
		condiz_ON_OFF:= HMI_cond[3],
		arc_level=> , 
		temp=> Tempz4, 
		funzione_1=> , 
		moviment_active=> , 
		condiz=> cononz4);
	luce_18(light_level:= , ADDR:= 18, MODE:= 0, daliBuffer:= DALI_BUFFER2);
	luce_19(light_level:= , ADDR:= 19, MODE:= 0, daliBuffer:= DALI_BUFFER2);
	luce_20(light_level:= , ADDR:= 20, MODE:= 0, daliBuffer:= DALI_BUFFER2);
	IF ulux_3.arc_level=0 THEN
		luce_17.light_level:=0;
		luce_18.light_level:=0;
		luce_19.light_level:=0;
		luce_20.light_level:=0;
	ELSIF ulux_3.funzione_1=1 THEN
		luce_17.light_level:=0;
		luce_18.light_level:=200;
		luce_19.light_level:=200;
		luce_20.light_level:=254;
	ELSIF ulux_3.funzione_1=0  THEN
		luce_17.light_level:=ulux_3.arc_level;
		luce_18.light_level:=ulux_3.arc_level;
		luce_19.light_level:=ulux_3.arc_level;
		luce_20.light_level:=ulux_3.arc_level;
	END_IF
	IF luce_20.light_level<>0 THEN
		meetingroom_active:=TRUE;
	ELSE
		meetingroom_active:=FALSE;
	END_IF
//Ufficio Tecnico Gruppo:5 ID:4
	ulux_4(
		ID:= 4, 
		luci_OFF:= luci_ufficio_off OR HMI_luci_off[4], 
		luci_ON:= HMI_luci_on[4], 
		time_delay:= , 
		condiz_ON_OFF:= HMI_cond[4],
		arc_level=> , 
		temp=> Tempz5, 
		funzione_1=> , 
		moviment_active=> , 
		condiz=> cononz5);
	group_5(light_level:= ulux_4.arc_level, ADDR:= 5, MODE:= 1, daliBuffer:= DALI_BUFFER2);
//Ufficio Produzione Gruppo:6 ID:5
	ulux_5(
		ID:= 5, 
		luci_OFF:= luci_ufficio_off OR HMI_luci_off[5], 
		luci_ON:= HMI_luci_on[5], 
		time_delay:= , 
		condiz_ON_OFF:= HMI_cond[5],
		arc_level=> , 
		temp=> Tempz6, 
		funzione_1=> , 
		moviment_active=> , 
		condiz=> cononz6);
	group_6(light_level:= ulux_5.arc_level, ADDR:= 6, MODE:= 1, daliBuffer:= DALI_BUFFER2);
//Locale Svago Gruppo:7 ID:6
	ulux_6(
		ID:= 6, 
		luci_OFF:= luci_ufficio_off OR HMI_luci_off[6],
		luci_ON:= HMI_luci_on[6], 
		time_delay:= , 
		condiz_ON_OFF:= HMI_cond[6],
		arc_level=> , 
		temp=> Tempz7, 
		funzione_1=> , 
		moviment_active=> , 
		condiz=> cononz7);
	group_7(light_level:= ulux_6.arc_level, ADDR:= 7, MODE:= 1, daliBuffer:= DALI_BUFFER2);
	//Server #16
		movimento_server(ID:=16#0199AF47, BAT_KO=> , LUX=> , Moviment=> );
		delay_luce_server(IN:= movimento_server.Moviment OR HMI_luce_server, PT:=T#2M , Q=> , ET=> );
		IF delay_luce_server.Q THEN
			luce_server.light_level:=254;
		ELSE
			luce_server.light_level:=0;
		END_IF
		luce_server(light_level:= , ADDR:=16 , MODE:=0 , daliBuffer:= DALI_BUFFER2);
	//Locale Stampante Gruppo:8 
		group_8(light_level:= gruppo8_arc_level, ADDR:= 8, MODE:= 1, daliBuffer:= DALI_BUFFER2);
	//Officina R&D Gruppo:9
		group_9(light_level:= gruppo9_arc_level, ADDR:= 9, MODE:= 1, daliBuffer:= DALI_BUFFER2);
	//Officina Gruppo:10
		group_10(light_level:= luci_capannone.light_level, ADDR:= 10, MODE:= 1, daliBuffer:= DALI_BUFFER2);

On_Off_luce1(
	pulsante:= pula3 OR pula4 OR KNX_p3, 
	ON:= , 
	OFF:=on_off_luce1.ADV , 
	up:=pulA1 , 
	down:=pulA2 , 
	light_level=> luce_1.light_level, 
	ADV=> );
luce_1(light_level:= , ADDR:= 1, MODE:= 0, daliBuffer:= DALI_BUFFER2);
On_Off_Gruppo0(
	pulsante:= pula3 OR knx_p1, 
	ON:= pulc1 OR puld1, 
	OFF:= on_off_gruppo0.ADV, 
	up:= pulb1 OR KNX_p2, 
	down:= pulb2 OR KNX_p4, 
	light_level=> gruppo0.light_level, 
	ADV=> );
gruppo0(light_level:=250 , ADDR:= , MODE:= 2, daliBuffer:= DALI_BUFFER1);

END_PROGRAM

// ---- POUs/ProjetcFB/EnO_TK_SR65_LI.TcPOU
FUNCTION_BLOCK EnO_TK_SR65_LI
VAR_INPUT
	ID: DWORD;
END_VAR
VAR_OUTPUT
	LUX: WORD;
	status: BOOL; (*TRUE = Low Voltage; False = Voltage OK*);
END_VAR
VAR
	READ: FB_Rec_Generic;
	POWER: DINT;
END_VAR

READ(
	str_KL6581:=enocean_buffer , 
	byNode:=1 , 
	dw_ID:=ID , 
	ar_Value=> , 
	by_Node=> , 
	by_STATE=> , 
	bReceive=> , 
	EnOceanTyp=> );

LUX:=read.ar_Value[1]*4;	
POWER:=TRUNC(read.ar_Value[3]/50);
IF power < 3  THEN
	status:=TRUE;
ELSE
	status:=FALSE;
END_IF

END_FUNCTION_BLOCK

// ---- POUs/ProjetcFB/ULUX_STD.TcPOU
FUNCTION_BLOCK ULUX_STD
VAR_INPUT
	ID: WORD;
	luci_OFF:BOOL; //segnale ad impulso
	luci_ON:BOOL; //segnale ad impulso
	time_delay:TIME;
	condiz_ON_OFF: INT; //segnale ad impulso
	dimmer_on: BOOL;
END_VAR
VAR_OUTPUT
	arc_level: BYTE;
	temp: UINT;
	funzione_1: INT;
	moviment_active:BOOL;
	condiz:INT;
	password1:INT;
	password2:INT;
	password3:INT;
	password4:INT;
END_VAR
VAR
	On_off_luce: FB_GET_ULUX_EDIT_VALUE;
	On_off_cond: FB_GET_ULUX_EDIT_VALUE;
	luce: INT;
	motion: BOOL;
	light_level: BYTE;
	Dimmer_luci: FB_GET_ULUX_EDIT_VALUE;
	Set_dimmer_luci: FB_SET_ULUX_EDIT_VALUE;
	dimmer: INT;
	puls_funz_1: FB_GET_ULUX_EDIT_VALUE;
	temperatura: FB_GET_ULUX_TEMPERATURE;
	movimento: FB_GET_ULUX_MOTIONSENSOR;
	lux: FB_GET_ULUX_LUX;
	val_lux: WORD;
	Set_light_off: FB_SET_ULUX_EDIT_VALUE;
	Set_light_on: FB_SET_ULUX_EDIT_VALUE;
	Set_cond_on: FB_SET_ULUX_EDIT_VALUE;
	Set_cond_off: FB_SET_ULUX_EDIT_VALUE;
	Set_estate: FB_SET_ULUX_EDIT_VALUE;
	Set_inverno: FB_SET_ULUX_EDIT_VALUE;
	puls_password1: FB_GET_ULUX_EDIT_VALUE;
	puls_password2: FB_GET_ULUX_EDIT_VALUE;
	puls_password3: FB_GET_ULUX_EDIT_VALUE;
	puls_password4: FB_GET_ULUX_EDIT_VALUE;
	val_light_off: INT :=0;
	val_light_ON: INT :=1;
	val_estate: INT :=1;
	val_inverno: INT :=0;
	val_condiz_ON: INT :=1;
	val_condiz_OFF: INT :=0;
	val_dimmer: INT;
	delay_moviment: TOF;
	mov_on: R_TRIG;
	mov_off: F_TRIG;
	HMI_levelperc: WSTRING;
	(*reset_luci: TON;
	val_dimmer_restart: INT :=220;
	Set_dimmer: FB_SET_ULUX_EDIT_VALUE;*)
END_VAR

//Accensione luci con ULUX
On_off_luce(
	iEditValue:= luce, 
	stCmdB:= ulux_buffer, 
	dwActorID:= (ID*10)+1, 
	bGetValue:= ,  
	bGetAfterReconnect:= TRUE, 
	bReceivedData=> , 
	dwRecFromSwitchID=> , 
	bBusy=> , 
	bError=> , 
	eErrUluxId=> );
//Dimmer luci con ULUX
Dimmer_luci(
	iEditValue:= dimmer, 
	stCmdB:= ulux_buffer, 
	dwActorID:= (ID*10)+2, 
	bGetValue:= , 
	bGetAfterReconnect:= TRUE, 
	bReceivedData=> , 
	dwRecFromSwitchID=> , 
	bBusy=> , 
	bError=> , 
	eErrUluxId=> );
CASE dimmer OF
	0:light_level:=85;
	12:light_level:=93;
	24:light_level:=101;
	36:light_level:=109;
	48:light_level:=117;
	60:light_level:=125;
	72:light_level:=133;
	84:light_level:=141;
	96:light_level:=149;
	108:light_level:=157;
	120:light_level:=165;
	132:light_level:=173;
	144:light_level:=181;
	156:light_level:=189;
	168:light_level:=197;
	180:light_level:=205;
	192:light_level:=213;
	204:light_level:=221;
	216:light_level:=229;
	228:light_level:=237;
	240:light_level:=245;
	252:light_level:=254;
ELSE
	light_level:=254;
END_CASE
IF luce=0 THEN
	arc_level:=0;
ELSIF luce=1 THEN
	arc_level:=light_level;
END_IF
//Valore in percentuale livello luce
CASE arc_level OF
	0: HMI_levelperc:="0 %";
	85: HMI_levelperc:="5 %";
	93: HMI_levelperc:="9 %";
	101: HMI_levelperc:="14 %";
	109: HMI_levelperc:="18 %";
	117: HMI_levelperc:="23 %";
	125: HMI_levelperc:="27 %";
	133: HMI_levelperc:="32 %";
	141: HMI_levelperc:="36 %";
	149: HMI_levelperc:="41 %";
	157: HMI_levelperc:="45 %";
	165: HMI_levelperc:="50 %";
	173: HMI_levelperc:="54 %";
	181: HMI_levelperc:="59 %";
	189: HMI_levelperc:="63 %";
	197: HMI_levelperc:="68 %";
	205: HMI_levelperc:="72 %";
	213: HMI_levelperc:="77 %";
	221: HMI_levelperc:="81 %";
	229: HMI_levelperc:="86 %";
	237: HMI_levelperc:="90 %";
	245: HMI_levelperc:="95 %";
	254: HMI_levelperc:="100 %";
END_CASE
//SET dimmer luci da PLC
Set_dimmer_luci(
	iEditValue:= val_dimmer, 
	stCmdB:= ulux_buffer, 
	dwActorID:= (ID*10)+2, 
	bSetValue:= dimmer_on, 
	bSetAfterReconnect:= (*true*), 
	bBusy=> , 
	bError=> , 
	eErrUluxId=> );
//Pulsante funzione 1
puls_funz_1(
	iEditValue:= funzione_1, 
	stCmdB:= ulux_buffer, 
	dwActorID:= (ID*10)+4, 
	bGetValue:= , 
	bGetAfterReconnect:= , 
	bReceivedData=> , 
	dwRecFromSwitchID=> , 
	bBusy=> , 
	bError=> , 
	eErrUluxId=> );
//Temperatura da ULUX
temperatura(
	stCmdB:= ulux_buffer, 
	dwSwitchID:= (ID+1), 
	bEnable:= TRUE, 
	bGetTemperature:= , 
	bTemperaturValid=> , 
	rTemperature=> , 
	bReceivedData=> , 
	bBusy=> , 
	bError=> , 
	eErrUluxId=> );
temp:= REAL_TO_UINT(temperatura.rTemperature*10);
//Movimento da ULUX
movimento(
	stCmdB:= ulux_buffer, 
	dwSwitchID:= (ID+1), 
	bEnable:= TRUE, 
	bMotionSensorOn=> , 
	bMotionDetect=> motion, 
	bReceivedData=> , 
	bBusy=> , 
	bError=> , 
	eErrUluxId=> );

delay_moviment(IN:= motion, PT:= time_delay, Q=>moviment_active , ET=> );

mov_on(CLK:=motion , Q=> );
mov_off(CLK:=delay_moviment.Q , Q=> );
//Lux da ULUX
lux(
	stCmdB:= ulux_buffer, 
	dwSwitchID:= (ID+1), 
	bEnable:= TRUE, 
	bGetLux:= , 
	bLuxValid=> , 
	wLux=> val_lux, 
	bReceivedData=> , 
	bBusy=> , 
	bError=> , 
	eErrUluxId=> );
IF luce=1 THEN
	HMI_luci_on[ID]:=TRUE;
	HMI_luci_off[ID]:=FALSE;
ELSE
	HMI_luci_on[ID]:=FALSE;
	HMI_luci_off[ID]:=TRUE;
END_IF
//SET spegni luci da PLC
Set_light_off(
	iEditValue:= val_light_off, 
	stCmdB:= ulux_buffer, 
	dwActorID:= (ID*10)+1, 
	bSetValue:= luci_off OR mov_off.Q, 
	bSetAfterReconnect:= (*true*), 
	bBusy=> , 
	bError=> , 
	eErrUluxId=> );
//SET accendi luci da PLC
Set_light_on(
	iEditValue:= val_light_on, 
	stCmdB:= ulux_buffer, 
	dwActorID:= (ID*10)+1, 
	bSetValue:= mov_on.Q OR LUCI_ON, 
	bSetAfterReconnect:= TRUE, 
	bBusy=> , 
	bError=> , 
	eErrUluxId=> );
//SET immagine estate su ULUX da PLC
Set_estate(
	iEditValue:= val_estate , 
	stCmdB:= ulux_buffer, 
	dwActorID:= (ID*10)+5, 
	bSetValue:= estate, 
	bSetAfterReconnect:= , 
	bBusy=> , 
	bError=> , 
	eErrUluxId=> );	
//SET immagine inverno su ULUX da PLC
Set_inverno(
	iEditValue:= val_inverno , 
	stCmdB:= ulux_buffer, 
	dwActorID:= (ID*10)+5, 
	bSetValue:= inverno, 
	bSetAfterReconnect:= , 
	bBusy=> , 
	bError=> , 
	eErrUluxId=> );
IF OFFICE_VHAC_EI THEN
	estate:=TRUE;
	inverno:=FALSE;
ELSIF NOT OFFICE_VHAC_EI THEN
	inverno:=TRUE;
	estate:=FALSE;
END_IF

//Condizionatori ON-OFF con ULUX
On_off_cond(
	iEditValue:= condiz, 
	stCmdB:= ulux_buffer, 
	dwActorID:= (ID*10)+5, 
	bGetValue:= , 
	bGetAfterReconnect:= , 
	bReceivedData=> , 
	dwRecFromSwitchID=> , 
	bBusy=> , 
	bError=> , 
	eErrUluxId=> );
//Spegnimento aria condizionata e cambiamento stato ULUX con allarme
IF allarme_Attivo<>0 (*allarme*) THEN
	condiz:=0;
END_IF
//SET condizionatori ON da PLC
Set_cond_on(
	iEditValue:= val_condiz_ON, 
	stCmdB:= ulux_buffer, 
	dwActorID:= (ID*10)+5, 
	bSetValue:= condiz_ON_OFF=1, 
	bSetAfterReconnect:= (*true*), 
	bBusy=> , 
	bError=> , 
	eErrUluxId=> );
IF mov_off.Q THEN
	condiz_ON_OFF:=0;
END_IF
(*IF condiz=1 THEN
	HMI_cond[ID]:=1;
ELSE
	HMI_cond[ID]:=0;
END_IF*)
//SET condizionatori OFF da PLC
Set_cond_off(
	iEditValue:= val_condiz_OFF, 
	stCmdB:= ulux_buffer, 
	dwActorID:= (ID*10)+5, 
	bSetValue:= allarme_Attivo<>0(*allarme*) OR condiz_ON_OFF=0, 
	bSetAfterReconnect:= (*true*), 
	bBusy=> , 
	bError=> , 
	eErrUluxId=> );
	
(*var_plc:=FALSE;
reset_luci(IN:= NOT var_plc, PT:= T#20S, Q=> , ET=> );
if reset_luci.Q then
	var_plc:=true;
END_IF
//SET imposta LUX al riavvio del PLC
Set_dimmer(
	iEditValue:= val_dimmer_restart, 
	stCmdB:= ulux_buffer, 
	dwActorID:= (ID*10)+1, 
	bSetValue:= reset_luci.Q, 
	bSetAfterReconnect:= TRUE, 
	bBusy=> , 
	bError=> , 
	eErrUluxId=> );*)
	
(*//Pulsante numeri password
puls_password1(
	iEditValue:= password1, 
	stCmdB:= ulux_buffer, 
	dwActorID:= (ID*10)+6, 
	bGetValue:=, 
	bGetAfterReconnect:= , 
	bBusy=> , 
	bError=> , 
	eErrUluxId=> );
puls_password2(
	iEditValue:= password2, 
	stCmdB:= ulux_buffer, 
	dwActorID:= (ID*10)+7, 
	bGetValue:=, 
	bGetAfterReconnect:= , 
	bBusy=> , 
	bError=> , 
	eErrUluxId=> );
puls_password3(
	iEditValue:= password3, 
	stCmdB:= ulux_buffer, 
	dwActorID:= (ID*10)+8, 
	bGetValue:=, 
	bGetAfterReconnect:= , 
	bBusy=> , 
	bError=> , 
	eErrUluxId=> );
puls_password4(
	iEditValue:= password4, 
	stCmdB:= ulux_buffer, 
	dwActorID:= (ID*10)+9, 
	bGetValue:=, 
	bGetAfterReconnect:= , 
	bBusy=> , 
	bError=> , 
	eErrUluxId=> );*)

END_FUNCTION_BLOCK

// ---- POUs/ULUX.TcPOU
PROGRAM ULUX
VAR
	ulux_comm: FB_ULUX_COM;
	umidita_riunioni: FB_GET_ULUX_HUMIDITY;
	prossimita_riunioni: FB_GET_ULUX_PROXIMITYSENSOR;
	on_off_riunioni: INT;
	dimmer1: INT;
	dimmer_riunioni: FB_GET_ULUX_EDIT_VALUE;
	on_off_luce: FB_GET_ULUX_EDIT_VALUE;
	luce: Dali_arcpower_control;
	luce_PROIETTORE: Dali_arcpower_control;
	luce_dimmer: Dali_arcpower_control;
	temperatura: REAL;
	umidita: REAL;
	lux: REAL;
	on_off_proiettore: FB_GET_ULUX_EDIT_VALUE;
	proiettore: INT;
	Cambio_Pagina_password: FB_SET_ULUX_PAGE;
	Cambio_Pagina_main: FB_SET_ULUX_PAGE;
	pippo: BOOL;
	password_ok: BOOL;
	t_password: TON;
	password: ULUX_STD;
	ledstate: FB_SET_ULUX_LEDSTATE;
	minnie1: BOOL;
END_VAR

//Comunicazione ulux
ulux_comm(
	bEnableCom:= TRUE, 
	sSrvNetId:= '5.37.99.190.1.1',
	sHostIpAddr:= '192.168.60.120', 
	sSubNetMask:= '255.255.255.0', 
	tStartUpDelay:= T#15S, 
	stTimestruct:= tempo_ulux, 
	stCmdB:= ulux_buffer, 
	bComActiv=> , 
	bBusy=> , 
	bError=> , 
	nErrId=> , 
	eErrUluxId=> );
	
//Cambio pagine ulux
Cambio_Pagina_password(
	stCmdB:= ulux_buffer, 
	dwSwitchID:= 5, 
	bSetPage:= , 
	byPageNumber:= 4, 
	bBusy=> , 
	bError=> , 
	eErrUluxId=> );
Cambio_Pagina_main(
	stCmdB:= ulux_buffer, 
	dwSwitchID:= 5, 
	bSetPage:= , 
	byPageNumber:= 2, 
	bBusy=> , 
	bError=> , 
	eErrUluxId=> );
IF pippo THEN
	cambio_pagina_password.bSetPage:=TRUE;
END_IF
password(
	ID:= 4, 
	luci_OFF:= , 
	luci_ON:= , 
	time_delay:= , 
	arc_level=> , 
	temp=> , 
	funzione_1=> , 
	moviment_active=> , 
	condiz=> , 
	password1=> , 
	password2=> , 
	password3=> , 
	password4=> );
IF password.password1=2 AND password.password2=7 AND password.password3=3 AND password.password4=8 THEN
	password_ok:=TRUE;
ELSE
	password_ok:=FALSE;
END_IF
IF password_ok THEN
	cambio_pagina_password.bSetPage:=FALSE;
	cambio_pagina_main.bSetPage:=TRUE;
	pippo:=FALSE;
END_IF
t_password(IN:= password_ok, PT:= T#5S, Q=> , ET=> );
IF t_password.Q THEN
	password_ok:=FALSE;
	cambio_pagina_main.bSetPage:=FALSE;
END_IF

ledstate(
	stCmdB:= ulux_buffer, 
	dwActorID:= 53, 
	bSetLed:= minnie1, 
	eLedBlink1:= 4, 
	eLedColor1:= 1, 
	eLedBlink2:= 4, 
	eLedColor2:= 2, 
	eLedBlink3:= 4, 
	eLedColor3:= 3, 
	eLedBlink4:= 4, 
	eLedColor4:= 4, 
	bLedOverride1:= , 
	bLedOverride2:= , 
	bLedOverride3:= , 
	bLedOverride4:= , 
	bSendAutoByChange:= , 
	tMinDelay:= , 
	bBusy=> , 
	bError=> , 
	eErrUluxId=> );
	
(*//Rilevamento umidità ulux
umidita_riunioni(
	stCmdB:= ulux_buffer, 
	dwSwitchID:= gvl_ulux.PROJEKT_ULUX_SWITCH_RIUNIONI_ID, 
	bEnable:= TRUE, 
	bGetHumidity:= , 
	bHumidityValid=> , 
	rHumidity=> , 
	bReceivedData=> , 
	bBusy=> , 
	bError=> , 
	eErrUluxId=> );
//Sensore di prossimità ulux
prossimita_riunioni(
	stCmdB:= ulux_buffer, 
	dwSwitchID:= gvl_ulux.PROJEKT_ULUX_SWITCH_RIUNIONI_ID, 
	bEnable:= TRUE, 
	bProximitySensorValid=> , 
	bObjektNearly=> , 
	bReceivedData=> , 
	bBusy=> , 
	bError=> , 
	eErrUluxId=> );
//Accensione luce sala riunioni
on_off_luce(
	iEditValue:= on_off_riunioni, 
	stCmdB:= ulux_buffer, 
	dwActorID:= gvl_ulux.AKTOREN_ONOFF_LUCE_ID, 
	bGetValue:= , 
	bGetAfterReconnect:= , 
	bReceivedData=> , 
	dwRecFromSwitchID=> , 
	bBusy=> , 
	bError=> , 
	eErrUluxId=> );
IF on_off_riunioni=1 THEN
	luce.light_level:=luce_dimmer.light_level;
ELSE
	luce.light_level:=0;
END_IF
luce(light_level:= , ADDR:= 32, MODE:= 0, daliBuffer:= dali_buffer2);
temperatura:=temp_riunioni.rTemperature;
umidita:=umidita_riunioni.rHumidity;
lux:=lux_riunioni.wLux;
//Modalità proiettore
on_off_proiettore(
	iEditValue:= proiettore, 
	stCmdB:= ulux_buffer, 
	dwActorID:= gvl_ulux.AKTOREN_PROIETTORE_ID, 
	bGetValue:= , 
	bGetAfterReconnect:= , 
	bReceivedData=> , 
	dwRecFromSwitchID=> , 
	bBusy=> , 
	bError=> , 
	eErrUluxId=> );
luce_proiettore(light_level:= , ADDR:= 32, MODE:= 0, daliBuffer:= dali_buffer2);
IF proiettore=1 THEN
	luce_proiettore.light_level:=254;
ELSE
	luce_proiettore.light_level:=0;
END_IF*)

END_PROGRAM

// ---- POUs/KNX.TcPOU
PROGRAM KNX
VAR
	KNX_COMM: KL6301;
	KL6301_PHYS_ADDR: EIB_PHYS_ADDR;
	KNX_FILTERS: ARRAY [1..8] OF EIB_GROUP_FILTER;
	KNX_BUFFER: EIB_REC;
	KNX_IN AT %I*: ARRAY [1..24] OF BYTE;
	KNX_OUT AT %Q*: ARRAY [1..24] OF BYTE;
	Leggi_Temp: EIB_2OCTET_FLOAT_REC;
	Leggi_luxf: EIB_2OCTET_FLOAT_REC;
	Leggi_luxR: EIB_2OCTET_FLOAT_REC;
	Leggi_luxL: EIB_2OCTET_FLOAT_REC;
	Leggi_wind: EIB_2OCTET_FLOAT_REC;
	Leggi_rain:EIB_BIT_REC;
	Leggi_stato_temp: EIB_BIT_REC;
	GROUP_ADDR_MAIN: INT;
	G_t1: EIB_GROUP_ADDR;
	G_luxF: EIB_GROUP_ADDR;
	G_luxR: EIB_GROUP_ADDR;
	G_luxL: EIB_GROUP_ADDR;
	G_wind: EIB_GROUP_ADDR;
	G_rain: EIB_GROUP_ADDR;
	G_stato_temp: EIB_GROUP_ADDR;
	G_t0: EIB_GROUP_ADDR;
	G_P1: EIB_GROUP_ADDR;
	G_P2: EIB_GROUP_ADDR;
	G_P3: EIB_GROUP_ADDR;
	G_P4: EIB_GROUP_ADDR;
	Leggi_p1:EIB_BIT_REC;
	Leggi_p2:EIB_BIT_REC;
	Leggi_p3:EIB_BIT_REC;
	Leggi_p4:EIB_BIT_REC;
	Leggi_Temp0: EIB_2OCTET_FLOAT_REC;
END_VAR

KL6301_PHYS_ADDR.Area:=1;
KL6301_PHYS_ADDR.Device:=1;
KL6301_PHYS_ADDR.Line:=254;

KNX_FILTERS[1].GROUP_ADDR.MAIN:=0;
KNX_FILTERS[1].GROUP_ADDR.SUB_MAIN:=0;
KNX_FILTERS[1].GROUP_ADDR.NUMBER:=1;
KNX_FILTERS[1].GROUP_LEN:=32;


KNX_COMM(
	bActivate:=TRUE , 
	idx:= 1, 
	EIB_PHYS_ADDR:= KL6301_PHYS_ADDR, 
	EIB_GROUP_FILTER:=KNX_FILTERS, 
	iMode:= , 
	bActive=> , 
	bReady=> , 
	bError=> , 
	iErrorId=> , 
	str_Data_Rec=>KNX_BUFFER , 
	KL6301_IN:=KNX_IN , 
	KL6301_OUT:= KNX_OUT);
// Indirizzo Temperatura Esterna
	G_T1.MAIN:=0;
	G_T1.SUB_MAIN:=0;
	G_T1.NUMBER:=2;
// Indirizzo lux Frontale	
	G_luxF.MAIN:=0;
	G_luxF.SUB_MAIN:=0;
	G_luxF.NUMBER:=3;
// Indirizzo lux Frontale	
	G_luxR.MAIN:=0;
	G_luxR.SUB_MAIN:=0;
	G_luxR.NUMBER:=4;
// Indirizzo lux Frontale	
	G_luxL.MAIN:=0;
	G_luxL.SUB_MAIN:=0;
	G_luxL.NUMBER:=5;	
// Indirizzo Sensore Vento
	G_wind.MAIN:=0;
	G_wind.SUB_MAIN:=0;
	G_wind.NUMBER:=6;
// Indirizzo sensore pioggia
	G_rain.MAIN:=0;
	G_rain.SUB_MAIN:=0;
	G_rain.NUMBER:=7;	
// Indirizzo temperatura interna
	G_t0.MAIN:=0;
	G_t0.SUB_MAIN:=0;
	G_t0.NUMBER:=1;	
// Indirizzo pulsante1
	G_p1.MAIN:=0;
	G_p1.SUB_MAIN:=0;
	G_p1.NUMBER:=9;	
// Indirizzo pulsante2
	G_p2.MAIN:=0;
	G_p2.SUB_MAIN:=0;
	G_p2.NUMBER:=10;	
// Indirizzo pulsante3
	G_p3.MAIN:=0;
	G_p3.SUB_MAIN:=0;
	G_p3.NUMBER:=11;	
// Indirizzo pulsante4
	G_p4.MAIN:=0;
	G_p4.SUB_MAIN:=0;
	G_p4.NUMBER:=12;	

	Leggi_rain(Group_Address:= G_rain, strData_Rec:=KNX_BUFFER , bDataReceive=> , bData=>RAIN );
	Leggi_Temp(Group_Address:=G_t1 , strData_Rec:=KNX_BUFFER , bDataReceive=> , rData=>Temp_OUTSIDE );
	Leggi_luxf(Group_Address:=G_luxf, strData_Rec:=KNX_BUFFER , bDataReceive=> , rData=>LUX_OUTSIDEF);
	Leggi_luxR(Group_Address:=G_luxR, strData_Rec:=KNX_BUFFER , bDataReceive=> , rData=>LUX_OUTSIDER );
	Leggi_luxL(Group_Address:=G_luxL, strData_Rec:=KNX_BUFFER , bDataReceive=> , rData=>LUX_OUTSIDEL );
	Leggi_wind(Group_Address:=G_wind, strData_Rec:=KNX_BUFFER , bDataReceive=> , rData=>wind_speed );
	Leggi_p1(Group_Address:= G_p1, strData_Rec:=KNX_BUFFER , bDataReceive=> , bData=>knx_p1);
	Leggi_p2(Group_Address:= G_p2, strData_Rec:=KNX_BUFFER , bDataReceive=> , bData=>knx_p2 );
	Leggi_p3(Group_Address:= G_p3, strData_Rec:=KNX_BUFFER , bDataReceive=> , bData=>knx_p3 );
	Leggi_p4(Group_Address:= G_p4, strData_Rec:=KNX_BUFFER , bDataReceive=> , bData=>knx_p4 );
	Leggi_Temp0(Group_Address:=G_t0 , strData_Rec:=KNX_BUFFER , bDataReceive=> , rData=>Temp_INSIDE );
	Leggi_stato_temp(Group_Address:=G_stato_temp, strData_Rec:=KNX_BUFFER , bDataReceive=> , bData=>stato_temp );

END_PROGRAM

// ---- POUs/Alarm.TcPOU
PROGRAM Alarm
VAR
	Timer_allarme: TON;
	allarme_tamper:BOOL;
	Timer_Sirena: TP;
	alarm_service: BOOL;
	rilevato_movimento: BOOL;
	rilevata_manomissione: BOOL;
	allarme_scattato: BOOL;
	SR_ainterno: SR;
	SR_afronte: SR;
	SR_aretro: SR;
	SR_asx: SR;
	SR_allarme: SR;
	SR_atamper: SR;
	SR_mensa: SR;
	SR_ingresso: SR;
	SR_tecnico: SR;
	
	F1_trig: F_TRIG;
	F2_trig: F_TRIG;
	F3_trig: F_TRIG;
	F4_trig: F_TRIG;
	F5_trig: F_TRIG;
	S1_trig: F_TRIG;
	S2_trig: F_TRIG;
	R1_trig: F_TRIG;
	R2_trig: F_TRIG;
	R3_trig: F_TRIG;
	R4_trig: F_TRIG;
	R5_trig: F_TRIG;
	D1_trig: F_TRIG;
	C1_trig: F_TRIG;
	C2_trig: F_TRIG;
	C3_trig: F_TRIG;
	U1_trig: F_TRIG;
	U2_trig: F_TRIG;
	U3_trig: F_TRIG;

